Fanuc TP program (LS listing): LOWWALL.LS

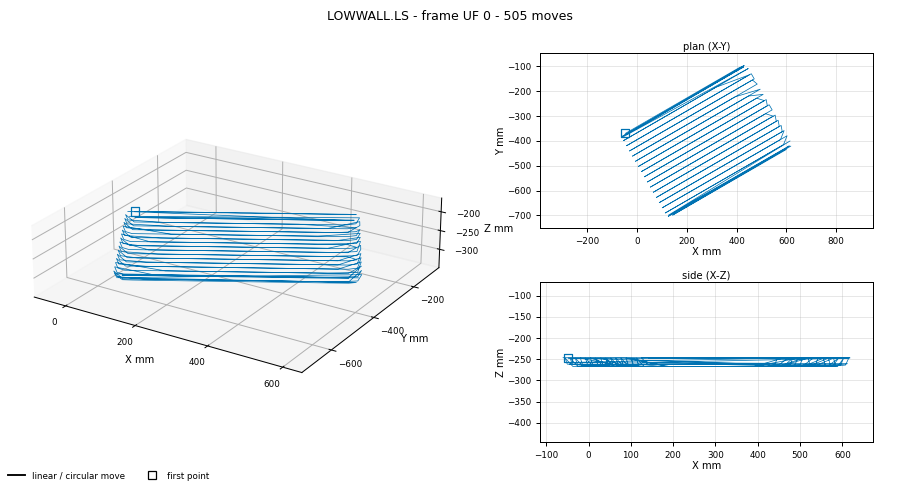
[picture p0: tool path of LOWWALL.LS in frame UF 0, 505 of 505 moves have a stored position in this frame; points joined in program order, loops and branches not executed]
/PROG  LOWWALL.LS
/ATTR
OWNER       = MNEDITOR;
COMMENT     = "";
PROG_SIZE   = 636;
CREATE      = DATE 23-01-07  TIME 11:59:14;
MODIFIED    = DATE 23-01-07  TIME 12:02:18;
FILE_NAME   = ;
VERSION     = 0;
LINE_COUNT  = 4;
MEMORY_SIZE = 992;
PROTECT     = READ_WRITE;
TCD:  STACK_SIZE	= 0,
      TASK_PRIORITY	= 50,
      TIME_SLICE	= 0,
      BUSY_LAMP_OFF	= 0,
      ABORT_REQUEST	= 0,
      PAUSE_REQUEST	= 0;
DEFAULT_GROUP	= 1,*,*,*,*;
CONTROL_CODE	= 00000000 00000000;
/MN
   1:J P[1] 100% FINE    ;
   2:L P[2] 100mm/sec CNT0    ;
   3:L P[3] 100mm/sec CNT0    ;
   4:L P[4] 100mm/sec CNT0    ;
   5:L P[5] 100mm/sec CNT0    ;
   6:L P[6] 100mm/sec CNT0    ;
   7:L P[7] 100mm/sec CNT0    ;
   8:L P[8] 100mm/sec CNT0    ;
   9:L P[9] 100mm/sec CNT0    ;
   10:L P[10] 100mm/sec CNT0    ;
   11:L P[11] 100mm/sec CNT0    ;
   12:L P[12] 100mm/sec CNT0    ;
   13:L P[13] 100mm/sec CNT0    ;
   14:L P[14] 100mm/sec CNT0    ;
   15:L P[15] 100mm/sec CNT0    ;
   16:L P[16] 100mm/sec CNT0    ;
   17:L P[17] 100mm/sec CNT0    ;
   18:L P[18] 100mm/sec CNT0    ;
   19:L P[19] 100mm/sec CNT0    ;
   20:L P[20] 100mm/sec CNT0    ;
   21:L P[21] 100mm/sec CNT0    ;
   22:L P[22] 100mm/sec CNT0    ;
   23:L P[23] 100mm/sec CNT0    ;
   24:L P[24] 100mm/sec CNT0    ;
   25:L P[25] 100mm/sec CNT0    ;
   26:L P[26] 100mm/sec CNT0    ;
   27:L P[27] 100mm/sec CNT0    ;
   28:L P[28] 100mm/sec CNT0    ;
   29:L P[29] 100mm/sec CNT0    ;
   30:L P[30] 100mm/sec CNT0    ;
   31:L P[31] 100mm/sec CNT0    ;
   32:L P[32] 100mm/sec CNT0    ;
   33:L P[33] 100mm/sec CNT0    ;
   34:L P[34] 100mm/sec CNT0    ;
   35:L P[35] 100mm/sec CNT0    ;
   36:L P[36] 100mm/sec CNT0    ;
   37:L P[37] 100mm/sec CNT0    ;
   38:L P[38] 100mm/sec CNT0    ;
   39:L P[39] 100mm/sec CNT0    ;
   40:L P[40] 100mm/sec CNT0    ;
   41:L P[41] 100mm/sec CNT0    ;
   42:L P[42] 100mm/sec CNT0    ;
   43:L P[43] 100mm/sec CNT0    ;
   44:L P[44] 100mm/sec CNT0    ;
   45:L P[45] 100mm/sec CNT0    ;
   46:L P[46] 100mm/sec CNT0    ;
   47:L P[47] 100mm/sec CNT0    ;
   48:L P[48] 100mm/sec CNT0    ;
   49:L P[49] 100mm/sec CNT0    ;
   50:L P[50] 100mm/sec CNT0    ;
   51:L P[51] 100mm/sec CNT0    ;
   52:L P[52] 100mm/sec CNT0    ;
   53:L P[53] 100mm/sec CNT0    ;
   54:L P[54] 100mm/sec CNT0    ;
   55:L P[55] 100mm/sec CNT0    ;
   56:L P[56] 100mm/sec CNT0    ;
   57:L P[57] 100mm/sec CNT0    ;
   58:L P[58] 100mm/sec CNT0    ;
   59:L P[59] 100mm/sec CNT0    ;
   60:L P[60] 100mm/sec CNT0    ;
   61:L P[61] 100mm/sec CNT0    ;
   62:L P[62] 100mm/sec CNT0    ;
   63:L P[63] 100mm/sec CNT0    ;
   64:L P[64] 100mm/sec CNT0    ;
   65:L P[65] 100mm/sec CNT0    ;
   66:L P[66] 100mm/sec CNT0    ;
   67:L P[67] 100mm/sec CNT0    ;
   68:L P[68] 100mm/sec CNT0    ;
   69:L P[69] 100mm/sec CNT0    ;
   70:L P[70] 100mm/sec CNT0    ;
   71:L P[71] 100mm/sec CNT0    ;
   72:L P[72] 100mm/sec CNT0    ;
   73:L P[73] 100mm/sec CNT0    ;
   74:L P[74] 100mm/sec CNT0    ;
   75:L P[75] 100mm/sec CNT0    ;
   76:L P[76] 100mm/sec CNT0    ;
   77:L P[77] 100mm/sec CNT0    ;
   78:L P[78] 100mm/sec CNT0    ;
   79:L P[79] 100mm/sec CNT0    ;
   80:L P[80] 100mm/sec CNT0    ;
   81:L P[81] 100mm/sec CNT0    ;
   82:L P[82] 100mm/sec CNT0    ;
   83:L P[83] 100mm/sec CNT0    ;
   84:L P[84] 100mm/sec CNT0    ;
   85:L P[85] 100mm/sec CNT0    ;
   86:L P[86] 100mm/sec CNT0    ;
   87:L P[87] 100mm/sec CNT0    ;
   88:L P[88] 100mm/sec CNT0    ;
   89:L P[89] 100mm/sec CNT0    ;
   90:L P[90] 100mm/sec CNT0    ;
   91:L P[91] 100mm/sec CNT0    ;
   92:L P[92] 100mm/sec CNT0    ;
   93:L P[93] 100mm/sec CNT0    ;
   94:L P[94] 100mm/sec CNT0    ;
   95:L P[95] 100mm/sec CNT0    ;
   96:L P[96] 100mm/sec CNT0    ;
   97:L P[97] 100mm/sec CNT0    ;
   98:L P[98] 100mm/sec CNT0    ;
   99:L P[99] 100mm/sec CNT0    ;
   100:L P[100] 100mm/sec CNT0    ;
   101:L P[101] 100mm/sec CNT0    ;
   102:L P[102] 100mm/sec CNT0    ;
   103:L P[103] 100mm/sec CNT0    ;
   104:L P[104] 100mm/sec CNT0    ;
   105:L P[105] 100mm/sec CNT0    ;
   106:L P[106] 100mm/sec CNT0    ;
   107:L P[107] 100mm/sec CNT0    ;
   108:L P[108] 100mm/sec CNT0    ;
   109:L P[109] 100mm/sec CNT0    ;
   110:L P[110] 100mm/sec CNT0    ;
   111:L P[111] 100mm/sec CNT0    ;
   112:L P[112] 100mm/sec CNT0    ;
   113:L P[113] 100mm/sec CNT0    ;
   114:L P[114] 100mm/sec CNT0    ;
   115:L P[115] 100mm/sec CNT0    ;
   116:L P[116] 100mm/sec CNT0    ;
   117:L P[117] 100mm/sec CNT0    ;
   118:L P[118] 100mm/sec CNT0    ;
   119:L P[119] 100mm/sec CNT0    ;
   120:L P[120] 100mm/sec CNT0    ;
   121:L P[121] 100mm/sec CNT0    ;
   122:L P[122] 100mm/sec CNT0    ;
   123:L P[123] 100mm/sec CNT0    ;
   124:L P[124] 100mm/sec CNT0    ;
   125:L P[125] 100mm/sec CNT0    ;
   126:L P[126] 100mm/sec CNT0    ;
   127:L P[127] 100mm/sec CNT0    ;
   128:L P[128] 100mm/sec CNT0    ;
   129:L P[129] 100mm/sec CNT0    ;
   130:L P[130] 100mm/sec CNT0    ;
   131:L P[131] 100mm/sec CNT0    ;
   132:L P[132] 100mm/sec CNT0    ;
   133:L P[133] 100mm/sec CNT0    ;
   134:L P[134] 100mm/sec CNT0    ;
   135:L P[135] 100mm/sec CNT0    ;
   136:L P[136] 100mm/sec CNT0    ;
   137:L P[137] 100mm/sec CNT0    ;
   138:L P[138] 100mm/sec CNT0    ;
   139:L P[139] 100mm/sec CNT0    ;
   140:L P[140] 100mm/sec CNT0    ;
   141:L P[141] 100mm/sec CNT0    ;
   142:L P[142] 100mm/sec CNT0    ;
   143:L P[143] 100mm/sec CNT0    ;
   144:L P[144] 100mm/sec CNT0    ;
   145:L P[145] 100mm/sec CNT0    ;
   146:L P[146] 100mm/sec CNT0    ;
   147:L P[147] 100mm/sec CNT0    ;
   148:L P[148] 100mm/sec CNT0    ;
   149:L P[149] 100mm/sec CNT0    ;
   150:L P[150] 100mm/sec CNT0    ;
   151:L P[151] 100mm/sec CNT0    ;
   152:L P[152] 100mm/sec CNT0    ;
   153:L P[153] 100mm/sec CNT0    ;
   154:L P[154] 100mm/sec CNT0    ;
   155:L P[155] 100mm/sec CNT0    ;
   156:L P[156] 100mm/sec CNT0    ;
   157:L P[157] 100mm/sec CNT0    ;
   158:L P[158] 100mm/sec CNT0    ;
   159:L P[159] 100mm/sec CNT0    ;
   160:L P[160] 100mm/sec CNT0    ;
   161:L P[161] 100mm/sec CNT0    ;
   162:L P[162] 100mm/sec CNT0    ;
   163:L P[163] 100mm/sec CNT0    ;
   164:L P[164] 100mm/sec CNT0    ;
   165:L P[165] 100mm/sec CNT0    ;
   166:L P[166] 100mm/sec CNT0    ;
   167:L P[167] 100mm/sec CNT0    ;
   168:L P[168] 100mm/sec CNT0    ;
   169:L P[169] 100mm/sec CNT0    ;
   170:L P[170] 100mm/sec CNT0    ;
   171:L P[171] 100mm/sec CNT0    ;
   172:L P[172] 100mm/sec CNT0    ;
   173:L P[173] 100mm/sec CNT0    ;
   174:L P[174] 100mm/sec CNT0    ;
   175:L P[175] 100mm/sec CNT0    ;
   176:L P[176] 100mm/sec CNT0    ;
   177:L P[177] 100mm/sec CNT0    ;
   178:L P[178] 100mm/sec CNT0    ;
   179:L P[179] 100mm/sec CNT0    ;
   180:L P[180] 100mm/sec CNT0    ;
   181:L P[181] 100mm/sec CNT0    ;
   182:L P[182] 100mm/sec CNT0    ;
   183:L P[183] 100mm/sec CNT0    ;
   184:L P[184] 100mm/sec CNT0    ;
   185:L P[185] 100mm/sec CNT0    ;
   186:L P[186] 100mm/sec CNT0    ;
   187:L P[187] 100mm/sec CNT0    ;
   188:L P[188] 100mm/sec CNT0    ;
   189:L P[189] 100mm/sec CNT0    ;
   190:L P[190] 100mm/sec CNT0    ;
   191:L P[191] 100mm/sec CNT0    ;
   192:L P[192] 100mm/sec CNT0    ;
   193:L P[193] 100mm/sec CNT0    ;
   194:L P[194] 100mm/sec CNT0    ;
   195:L P[195] 100mm/sec CNT0    ;
   196:L P[196] 100mm/sec CNT0    ;
   197:L P[197] 100mm/sec CNT0    ;
   198:L P[198] 100mm/sec CNT0    ;
   199:L P[199] 100mm/sec CNT0    ;
   200:L P[200] 100mm/sec CNT0    ;
   201:L P[201] 100mm/sec CNT0    ;
   202:L P[202] 100mm/sec CNT0    ;
   203:L P[203] 100mm/sec CNT0    ;
   204:L P[204] 100mm/sec CNT0    ;
   205:L P[205] 100mm/sec CNT0    ;
   206:L P[206] 100mm/sec CNT0    ;
   207:L P[207] 100mm/sec CNT0    ;
   208:L P[208] 100mm/sec CNT0    ;
   209:L P[209] 100mm/sec CNT0    ;
   210:L P[210] 100mm/sec CNT0    ;
   211:L P[211] 100mm/sec CNT0    ;
   212:L P[212] 100mm/sec CNT0    ;
   213:L P[213] 100mm/sec CNT0    ;
   214:L P[214] 100mm/sec CNT0    ;
   215:L P[215] 100mm/sec CNT0    ;
   216:L P[216] 100mm/sec CNT0    ;
   217:L P[217] 100mm/sec CNT0    ;
   218:L P[218] 100mm/sec CNT0    ;
   219:L P[219] 100mm/sec CNT0    ;
   220:L P[220] 100mm/sec CNT0    ;
   221:L P[221] 100mm/sec CNT0    ;
   222:L P[222] 100mm/sec CNT0    ;
   223:L P[223] 100mm/sec CNT0    ;
   224:L P[224] 100mm/sec CNT0    ;
   225:L P[225] 100mm/sec CNT0    ;
   226:L P[226] 100mm/sec CNT0    ;
   227:L P[227] 100mm/sec CNT0    ;
   228:L P[228] 100mm/sec CNT0    ;
   229:L P[229] 100mm/sec CNT0    ;
   230:L P[230] 100mm/sec CNT0    ;
   231:L P[231] 100mm/sec CNT0    ;
   232:L P[232] 100mm/sec CNT0    ;
   233:L P[233] 100mm/sec CNT0    ;
   234:L P[234] 100mm/sec CNT0    ;
   235:L P[235] 100mm/sec CNT0    ;
   236:L P[236] 100mm/sec CNT0    ;
   237:L P[237] 100mm/sec CNT0    ;
   238:L P[238] 100mm/sec CNT0    ;
   239:L P[239] 100mm/sec CNT0    ;
   240:L P[240] 100mm/sec CNT0    ;
   241:L P[241] 100mm/sec CNT0    ;
   242:L P[242] 100mm/sec CNT0    ;
   243:L P[243] 100mm/sec CNT0    ;
   244:L P[244] 100mm/sec CNT0    ;
   245:L P[245] 100mm/sec CNT0    ;
   246:L P[246] 100mm/sec CNT0    ;
   247:L P[247] 100mm/sec CNT0    ;
   248:L P[248] 100mm/sec CNT0    ;
   249:L P[249] 100mm/sec CNT0    ;
   250:L P[250] 100mm/sec CNT0    ;
   251:L P[251] 100mm/sec CNT0    ;
   252:L P[252] 100mm/sec CNT0    ;
   253:L P[253] 100mm/sec CNT0    ;
   254:L P[254] 100mm/sec CNT0    ;
   255:L P[255] 100mm/sec CNT0    ;
   256:L P[256] 100mm/sec CNT0    ;
   257:L P[257] 100mm/sec CNT0    ;
   258:L P[258] 100mm/sec CNT0    ;
   259:L P[259] 100mm/sec CNT0    ;
   260:L P[260] 100mm/sec CNT0    ;
   261:L P[261] 100mm/sec CNT0    ;
   262:L P[262] 100mm/sec CNT0    ;
   263:L P[263] 100mm/sec CNT0    ;
   264:L P[264] 100mm/sec CNT0    ;
   265:L P[265] 100mm/sec CNT0    ;
   266:L P[266] 100mm/sec CNT0    ;
   267:L P[267] 100mm/sec CNT0    ;
   268:L P[268] 100mm/sec CNT0    ;
   269:L P[269] 100mm/sec CNT0    ;
   270:L P[270] 100mm/sec CNT0    ;
   271:L P[271] 100mm/sec CNT0    ;
   272:L P[272] 100mm/sec CNT0    ;
   273:L P[273] 100mm/sec CNT0    ;
   274:L P[274] 100mm/sec CNT0    ;
   275:L P[275] 100mm/sec CNT0    ;
   276:L P[276] 100mm/sec CNT0    ;
   277:L P[277] 100mm/sec CNT0    ;
   278:L P[278] 100mm/sec CNT0    ;
   279:L P[279] 100mm/sec CNT0    ;
   280:L P[280] 100mm/sec CNT0    ;
   281:L P[281] 100mm/sec CNT0    ;
   282:L P[282] 100mm/sec CNT0    ;
   283:L P[283] 100mm/sec CNT0    ;
   284:L P[284] 100mm/sec CNT0    ;
   285:L P[285] 100mm/sec CNT0    ;
   286:L P[286] 100mm/sec CNT0    ;
   287:L P[287] 100mm/sec CNT0    ;
   288:L P[288] 100mm/sec CNT0    ;
   289:L P[289] 100mm/sec CNT0    ;
   290:L P[290] 100mm/sec CNT0    ;
   291:L P[291] 100mm/sec CNT0    ;
   292:L P[292] 100mm/sec CNT0    ;
   293:L P[293] 100mm/sec CNT0    ;
   294:L P[294] 100mm/sec CNT0    ;
   295:L P[295] 100mm/sec CNT0    ;
   296:L P[296] 100mm/sec CNT0    ;
   297:L P[297] 100mm/sec CNT0    ;
   298:L P[298] 100mm/sec CNT0    ;
   299:L P[299] 100mm/sec CNT0    ;
   300:L P[300] 100mm/sec CNT0    ;
   301:L P[301] 100mm/sec CNT0    ;
   302:L P[302] 100mm/sec CNT0    ;
   303:L P[303] 100mm/sec CNT0    ;
   304:L P[304] 100mm/sec CNT0    ;
   305:L P[305] 100mm/sec CNT0    ;
   306:L P[306] 100mm/sec CNT0    ;
   307:L P[307] 100mm/sec CNT0    ;
   308:L P[308] 100mm/sec CNT0    ;
   309:L P[309] 100mm/sec CNT0    ;
   310:L P[310] 100mm/sec CNT0    ;
   311:L P[311] 100mm/sec CNT0    ;
   312:L P[312] 100mm/sec CNT0    ;
   313:L P[313] 100mm/sec CNT0    ;
   314:L P[314] 100mm/sec CNT0    ;
   315:L P[315] 100mm/sec CNT0    ;
   316:L P[316] 100mm/sec CNT0    ;
   317:L P[317] 100mm/sec CNT0    ;
   318:L P[318] 100mm/sec CNT0    ;
   319:L P[319] 100mm/sec CNT0    ;
   320:L P[320] 100mm/sec CNT0    ;
   321:L P[321] 100mm/sec CNT0    ;
   322:L P[322] 100mm/sec CNT0    ;
   323:L P[323] 100mm/sec CNT0    ;
   324:L P[324] 100mm/sec CNT0    ;
   325:L P[325] 100mm/sec CNT0    ;
   326:L P[326] 100mm/sec CNT0    ;
   327:L P[327] 100mm/sec CNT0    ;
   328:L P[328] 100mm/sec CNT0    ;
   329:L P[329] 100mm/sec CNT0    ;
   330:L P[330] 100mm/sec CNT0    ;
   331:L P[331] 100mm/sec CNT0    ;
   332:L P[332] 100mm/sec CNT0    ;
   333:L P[333] 100mm/sec CNT0    ;
   334:L P[334] 100mm/sec CNT0    ;
   335:L P[335] 100mm/sec CNT0    ;
   336:L P[336] 100mm/sec CNT0    ;
   337:L P[337] 100mm/sec CNT0    ;
   338:L P[338] 100mm/sec CNT0    ;
   339:L P[339] 100mm/sec CNT0    ;
   340:L P[340] 100mm/sec CNT0    ;
   341:L P[341] 100mm/sec CNT0    ;
   342:L P[342] 100mm/sec CNT0    ;
   343:L P[343] 100mm/sec CNT0    ;
   344:L P[344] 100mm/sec CNT0    ;
   345:L P[345] 100mm/sec CNT0    ;
   346:L P[346] 100mm/sec CNT0    ;
   347:L P[347] 100mm/sec CNT0    ;
   348:L P[348] 100mm/sec CNT0    ;
   349:L P[349] 100mm/sec CNT0    ;
   350:L P[350] 100mm/sec CNT0    ;
   351:L P[351] 100mm/sec CNT0    ;
   352:L P[352] 100mm/sec CNT0    ;
   353:L P[353] 100mm/sec CNT0    ;
   354:L P[354] 100mm/sec CNT0    ;
   355:L P[355] 100mm/sec CNT0    ;
   356:L P[356] 100mm/sec CNT0    ;
   357:L P[357] 100mm/sec CNT0    ;
   358:L P[358] 100mm/sec CNT0    ;
   359:L P[359] 100mm/sec CNT0    ;
   360:L P[360] 100mm/sec CNT0    ;
   361:L P[361] 100mm/sec CNT0    ;
   362:L P[362] 100mm/sec CNT0    ;
   363:L P[363] 100mm/sec CNT0    ;
   364:L P[364] 100mm/sec CNT0    ;
   365:L P[365] 100mm/sec CNT0    ;
   366:L P[366] 100mm/sec CNT0    ;
   367:L P[367] 100mm/sec CNT0    ;
   368:L P[368] 100mm/sec CNT0    ;
   369:L P[369] 100mm/sec CNT0    ;
   370:L P[370] 100mm/sec CNT0    ;
   371:L P[371] 100mm/sec CNT0    ;
   372:L P[372] 100mm/sec CNT0    ;
   373:L P[373] 100mm/sec CNT0    ;
   374:L P[374] 100mm/sec CNT0    ;
   375:L P[375] 100mm/sec CNT0    ;
   376:L P[376] 100mm/sec CNT0    ;
   377:L P[377] 100mm/sec CNT0    ;
   378:L P[378] 100mm/sec CNT0    ;
   379:L P[379] 100mm/sec CNT0    ;
   380:L P[380] 100mm/sec CNT0    ;
   381:L P[381] 100mm/sec CNT0    ;
   382:L P[382] 100mm/sec CNT0    ;
   383:L P[383] 100mm/sec CNT0    ;
   384:L P[384] 100mm/sec CNT0    ;
   385:L P[385] 100mm/sec CNT0    ;
   386:L P[386] 100mm/sec CNT0    ;
   387:L P[387] 100mm/sec CNT0    ;
   388:L P[388] 100mm/sec CNT0    ;
   389:L P[389] 100mm/sec CNT0    ;
   390:L P[390] 100mm/sec CNT0    ;
   391:L P[391] 100mm/sec CNT0    ;
   392:L P[392] 100mm/sec CNT0    ;
   393:L P[393] 100mm/sec CNT0    ;
   394:L P[394] 100mm/sec CNT0    ;
   395:L P[395] 100mm/sec CNT0    ;
   396:L P[396] 100mm/sec CNT0    ;
   397:L P[397] 100mm/sec CNT0    ;
   398:L P[398] 100mm/sec CNT0    ;
   399:L P[399] 100mm/sec CNT0    ;
   400:L P[400] 100mm/sec CNT0    ;
   401:L P[401] 100mm/sec CNT0    ;
   402:L P[402] 100mm/sec CNT0    ;
   403:L P[403] 100mm/sec CNT0    ;
   404:L P[404] 100mm/sec CNT0    ;
   405:L P[405] 100mm/sec CNT0    ;
   406:L P[406] 100mm/sec CNT0    ;
   407:L P[407] 100mm/sec CNT0    ;
   408:L P[408] 100mm/sec CNT0    ;
   409:L P[409] 100mm/sec CNT0    ;
   410:L P[410] 100mm/sec CNT0    ;
   411:L P[411] 100mm/sec CNT0    ;
   412:L P[412] 100mm/sec CNT0    ;
   413:L P[413] 100mm/sec CNT0    ;
   414:L P[414] 100mm/sec CNT0    ;
   415:L P[415] 100mm/sec CNT0    ;
   416:L P[416] 100mm/sec CNT0    ;
   417:L P[417] 100mm/sec CNT0    ;
   418:L P[418] 100mm/sec CNT0    ;
   419:L P[419] 100mm/sec CNT0    ;
   420:L P[420] 100mm/sec CNT0    ;
   421:L P[421] 100mm/sec CNT0    ;
   422:L P[422] 100mm/sec CNT0    ;
   423:L P[423] 100mm/sec CNT0    ;
   424:L P[424] 100mm/sec CNT0    ;
   425:L P[425] 100mm/sec CNT0    ;
   426:L P[426] 100mm/sec CNT0    ;
   427:L P[427] 100mm/sec CNT0    ;
   428:L P[428] 100mm/sec CNT0    ;
   429:L P[429] 100mm/sec CNT0    ;
   430:L P[430] 100mm/sec CNT0    ;
   431:L P[431] 100mm/sec CNT0    ;
   432:L P[432] 100mm/sec CNT0    ;
   433:L P[433] 100mm/sec CNT0    ;
   434:L P[434] 100mm/sec CNT0    ;
   435:L P[435] 100mm/sec CNT0    ;
   436:L P[436] 100mm/sec CNT0    ;
   437:L P[437] 100mm/sec CNT0    ;
   438:L P[438] 100mm/sec CNT0    ;
   439:L P[439] 100mm/sec CNT0    ;
   440:L P[440] 100mm/sec CNT0    ;
   441:L P[441] 100mm/sec CNT0    ;
   442:L P[442] 100mm/sec CNT0    ;
   443:L P[443] 100mm/sec CNT0    ;
   444:L P[444] 100mm/sec CNT0    ;
   445:L P[445] 100mm/sec CNT0    ;
   446:L P[446] 100mm/sec CNT0    ;
   447:L P[447] 100mm/sec CNT0    ;
   448:L P[448] 100mm/sec CNT0    ;
   449:L P[449] 100mm/sec CNT0    ;
   450:L P[450] 100mm/sec CNT0    ;
   451:L P[451] 100mm/sec CNT0    ;
   452:L P[452] 100mm/sec CNT0    ;
   453:L P[453] 100mm/sec CNT0    ;
   454:L P[454] 100mm/sec CNT0    ;
   455:L P[455] 100mm/sec CNT0    ;
   456:L P[456] 100mm/sec CNT0    ;
   457:L P[457] 100mm/sec CNT0    ;
   458:L P[458] 100mm/sec CNT0    ;
   459:L P[459] 100mm/sec CNT0    ;
   460:L P[460] 100mm/sec CNT0    ;
   461:L P[461] 100mm/sec CNT0    ;
   462:L P[462] 100mm/sec CNT0    ;
   463:L P[463] 100mm/sec CNT0    ;
   464:L P[464] 100mm/sec CNT0    ;
   465:L P[465] 100mm/sec CNT0    ;
   466:L P[466] 100mm/sec CNT0    ;
   467:L P[467] 100mm/sec CNT0    ;
   468:L P[468] 100mm/sec CNT0    ;
   469:L P[469] 100mm/sec CNT0    ;
   470:L P[470] 100mm/sec CNT0    ;
   471:L P[471] 100mm/sec CNT0    ;
   472:L P[472] 100mm/sec CNT0    ;
   473:L P[473] 100mm/sec CNT0    ;
   474:L P[474] 100mm/sec CNT0    ;
   475:L P[475] 100mm/sec CNT0    ;
   476:L P[476] 100mm/sec CNT0    ;
   477:L P[477] 100mm/sec CNT0    ;
   478:L P[478] 100mm/sec CNT0    ;
   479:L P[479] 100mm/sec CNT0    ;
   480:L P[480] 100mm/sec CNT0    ;
   481:L P[481] 100mm/sec CNT0    ;
   482:L P[482] 100mm/sec CNT0    ;
   483:L P[483] 100mm/sec CNT0    ;
   484:L P[484] 100mm/sec CNT0    ;
   485:L P[485] 100mm/sec CNT0    ;
   486:L P[486] 100mm/sec CNT0    ;
   487:L P[487] 100mm/sec CNT0    ;
   488:L P[488] 100mm/sec CNT0    ;
   489:L P[489] 100mm/sec CNT0    ;
   490:L P[490] 100mm/sec CNT0    ;
   491:L P[491] 100mm/sec CNT0    ;
   492:L P[492] 100mm/sec CNT0    ;
   493:L P[493] 100mm/sec CNT0    ;
   494:L P[494] 100mm/sec CNT0    ;
   495:L P[495] 100mm/sec CNT0    ;
   496:L P[496] 100mm/sec CNT0    ;
   497:L P[497] 100mm/sec CNT0    ;
   498:L P[498] 100mm/sec CNT0    ;
   499:L P[499] 100mm/sec CNT0    ;
   500:L P[500] 100mm/sec CNT0    ;
   501:L P[501] 100mm/sec CNT0    ;
   502:L P[502] 100mm/sec CNT0    ;
   503:L P[503] 100mm/sec CNT0    ;
   504:L P[504] 100mm/sec CNT0    ;
   505:L P[505] 100mm/sec CNT0    ;
/POS
P[1]{
   GP1:
	UF : 0, UT : 6,		CONFIG : 'N U T, 0, 0, 0',
	X =  -47.550  mm,	Y =   -370.000  mm,	Z =   -247.494  mm,
	W =  90.000 deg,	P =   0.000 deg,	R =   90.000 deg
};
P[2]{
   GP1:
	UF : 0, UT : 6,		CONFIG : 'N U T, 0, 0, 0',
	X =  -26.618  mm,	Y =   -357.826  mm,	Z =   -247.507  mm,
	W =  90.000 deg,	P =   0.000 deg,	R =   90.000 deg
};
P[3]{
   GP1:
	UF : 0, UT : 6,		CONFIG : 'N U T, 0, 0, 0',
	X =  -5.744  mm,	Y =   -345.692  mm,	Z =   -247.310  mm,
	W =  90.000 deg,	P =   0.000 deg,	R =   90.000 deg
};
P[4]{
   GP1:
	UF : 0, UT : 6,		CONFIG : 'N U T, 0, 0, 0',
	X =  14.806  mm,	Y =   -333.821  mm,	Z =   -247.298  mm,
	W =  90.000 deg,	P =   0.000 deg,	R =   90.000 deg
};
P[5]{
   GP1:
	UF : 0, UT : 6,		CONFIG : 'N U T, 0, 0, 0',
	X =  35.704  mm,	Y =   -321.826  mm,	Z =   -247.469  mm,
	W =  90.000 deg,	P =   0.000 deg,	R =   90.000 deg
};
P[6]{
   GP1:
	UF : 0, UT : 6,		CONFIG : 'N U T, 0, 0, 0',
	X =  56.373  mm,	Y =   -309.892  mm,	Z =   -247.469  mm,
	W =  90.000 deg,	P =   0.000 deg,	R =   90.000 deg
};
P[7]{
   GP1:
	UF : 0, UT : 6,		CONFIG : 'N U T, 0, 0, 0',
	X =  77.152  mm,	Y =   -297.810  mm,	Z =   -247.265  mm,
	W =  90.000 deg,	P =   0.000 deg,	R =   90.000 deg
};
P[8]{
   GP1:
	UF : 0, UT : 6,		CONFIG : 'N U T, 0, 0, 0',
	X =  97.870  mm,	Y =   -285.956  mm,	Z =   -247.529  mm,
	W =  90.000 deg,	P =   0.000 deg,	R =   90.000 deg
};
P[9]{
   GP1:
	UF : 0, UT : 6,		CONFIG : 'N U T, 0, 0, 0',
	X =  118.697  mm,	Y =   -273.983  mm,	Z =   -247.655  mm,
	W =  90.000 deg,	P =   0.000 deg,	R =   90.000 deg
};
P[10]{
   GP1:
	UF : 0, UT : 6,		CONFIG : 'N U T, 0, 0, 0',
	X =  139.386  mm,	Y =   -261.886  mm,	Z =   -247.288  mm,
	W =  90.000 deg,	P =   0.000 deg,	R =   90.000 deg
};
P[11]{
   GP1:
	UF : 0, UT : 6,		CONFIG : 'N U T, 0, 0, 0',
	X =  160.242  mm,	Y =   -249.945  mm,	Z =   -247.534  mm,
	W =  90.000 deg,	P =   0.000 deg,	R =   90.000 deg
};
P[12]{
   GP1:
	UF : 0, UT : 6,		CONFIG : 'N U T, 0, 0, 0',
	X =  181.067  mm,	Y =   -237.977  mm,	Z =   -247.671  mm,
	W =  90.000 deg,	P =   0.000 deg,	R =   90.000 deg
};
P[13]{
   GP1:
	UF : 0, UT : 6,		CONFIG : 'N U T, 0, 0, 0',
	X =  202.067  mm,	Y =   -225.717  mm,	Z =   -247.343  mm,
	W =  90.000 deg,	P =   0.000 deg,	R =   90.000 deg
};
P[14]{
   GP1:
	UF : 0, UT : 6,		CONFIG : 'N U T, 0, 0, 0',
	X =  222.800  mm,	Y =   -213.811  mm,	Z =   -247.499  mm,
	W =  90.000 deg,	P =   0.000 deg,	R =   90.000 deg
};
P[15]{
   GP1:
	UF : 0, UT : 6,		CONFIG : 'N U T, 0, 0, 0',
	X =  243.481  mm,	Y =   -201.771  mm,	Z =   -247.259  mm,
	W =  90.000 deg,	P =   0.000 deg,	R =   90.000 deg
};
P[16]{
   GP1:
	UF : 0, UT : 6,		CONFIG : 'N U T, 0, 0, 0',
	X =  264.327  mm,	Y =   -189.775  mm,	Z =   -247.358  mm,
	W =  90.000 deg,	P =   0.000 deg,	R =   90.000 deg
};
P[17]{
   GP1:
	UF : 0, UT : 6,		CONFIG : 'N U T, 0, 0, 0',
	X =  284.999  mm,	Y =   -177.910  mm,	Z =   -247.531  mm,
	W =  90.000 deg,	P =   0.000 deg,	R =   90.000 deg
};
P[18]{
   GP1:
	UF : 0, UT : 6,		CONFIG : 'N U T, 0, 0, 0',
	X =  305.678  mm,	Y =   -165.935  mm,	Z =   -247.446  mm,
	W =  90.000 deg,	P =   0.000 deg,	R =   90.000 deg
};
P[19]{
   GP1:
	UF : 0, UT : 6,		CONFIG : 'N U T, 0, 0, 0',
	X =  326.574  mm,	Y =   -153.899  mm,	Z =   -247.516  mm,
	W =  90.000 deg,	P =   0.000 deg,	R =   90.000 deg
};
P[20]{
   GP1:
	UF : 0, UT : 6,		CONFIG : 'N U T, 0, 0, 0',
	X =  347.161  mm,	Y =   -142.012  mm,	Z =   -247.515  mm,
	W =  90.000 deg,	P =   0.000 deg,	R =   90.000 deg
};
P[21]{
   GP1:
	UF : 0, UT : 6,		CONFIG : 'N U T, 0, 0, 0',
	X =  368.204  mm,	Y =   -129.821  mm,	Z =   -247.414  mm,
	W =  90.000 deg,	P =   0.000 deg,	R =   90.000 deg
};
P[22]{
   GP1:
	UF : 0, UT : 6,		CONFIG : 'N U T, 0, 0, 0',
	X =  389.245  mm,	Y =   -117.683  mm,	Z =   -247.441  mm,
	W =  90.000 deg,	P =   0.000 deg,	R =   90.000 deg
};
P[23]{
   GP1:
	UF : 0, UT : 6,		CONFIG : 'N U T, 0, 0, 0',
	X =  409.743  mm,	Y =   -105.850  mm,	Z =   -247.448  mm,
	W =  90.000 deg,	P =   0.000 deg,	R =   90.000 deg
};
P[24]{
   GP1:
	UF : 0, UT : 6,		CONFIG : 'N U T, 0, 0, 0',
	X =  430.442  mm,	Y =   -96.886  mm,	Z =   -246.914  mm,
	W =  90.000 deg,	P =   0.000 deg,	R =   90.000 deg
};
P[25]{
   GP1:
	UF : 0, UT : 6,		CONFIG : 'N U T, 0, 0, 0',
	X =  -60.479  mm,	Y =   -382.088  mm,	Z =   -246.235  mm,
	W =  90.000 deg,	P =   0.000 deg,	R =   90.000 deg
};
P[26]{
   GP1:
	UF : 0, UT : 6,		CONFIG : 'N U T, 0, 0, 0',
	X =  412.489  mm,	Y =   -110.415  mm,	Z =   -261.820  mm,
	W =  90.000 deg,	P =   0.000 deg,	R =   90.000 deg
};
P[27]{
   GP1:
	UF : 0, UT : 6,		CONFIG : 'N U T, 0, 0, 0',
	X =  370.834  mm,	Y =   -134.410  mm,	Z =   -261.664  mm,
	W =  90.000 deg,	P =   0.000 deg,	R =   90.000 deg
};
P[28]{
   GP1:
	UF : 0, UT : 6,		CONFIG : 'N U T, 0, 0, 0',
	X =  350.053  mm,	Y =   -146.501  mm,	Z =   -261.826  mm,
	W =  90.000 deg,	P =   0.000 deg,	R =   90.000 deg
};
P[29]{
   GP1:
	UF : 0, UT : 6,		CONFIG : 'N U T, 0, 0, 0',
	X =  329.297  mm,	Y =   -158.443  mm,	Z =   -261.826  mm,
	W =  90.000 deg,	P =   0.000 deg,	R =   90.000 deg
};
P[30]{
   GP1:
	UF : 0, UT : 6,		CONFIG : 'N U T, 0, 0, 0',
	X =  287.613  mm,	Y =   -182.494  mm,	Z =   -261.786  mm,
	W =  90.000 deg,	P =   0.000 deg,	R =   90.000 deg
};
P[31]{
   GP1:
	UF : 0, UT : 6,		CONFIG : 'N U T, 0, 0, 0',
	X =  267.068  mm,	Y =   -194.329  mm,	Z =   -261.729  mm,
	W =  90.000 deg,	P =   0.000 deg,	R =   90.000 deg
};
P[32]{
   GP1:
	UF : 0, UT : 6,		CONFIG : 'N U T, 0, 0, 0',
	X =  246.212  mm,	Y =   -206.455  mm,	Z =   -261.878  mm,
	W =  90.000 deg,	P =   0.000 deg,	R =   90.000 deg
};
P[33]{
   GP1:
	UF : 0, UT : 6,		CONFIG : 'N U T, 0, 0, 0',
	X =  225.417  mm,	Y =   -218.435  mm,	Z =   -261.779  mm,
	W =  90.000 deg,	P =   0.000 deg,	R =   90.000 deg
};
P[34]{
   GP1:
	UF : 0, UT : 6,		CONFIG : 'N U T, 0, 0, 0',
	X =  184.036  mm,	Y =   -242.349  mm,	Z =   -261.866  mm,
	W =  90.000 deg,	P =   0.000 deg,	R =   90.000 deg
};
P[35]{
   GP1:
	UF : 0, UT : 6,		CONFIG : 'N U T, 0, 0, 0',
	X =  162.951  mm,	Y =   -254.466  mm,	Z =   -261.727  mm,
	W =  90.000 deg,	P =   0.000 deg,	R =   90.000 deg
};
P[36]{
   GP1:
	UF : 0, UT : 6,		CONFIG : 'N U T, 0, 0, 0',
	X =  142.127  mm,	Y =   -266.540  mm,	Z =   -261.832  mm,
	W =  90.000 deg,	P =   0.000 deg,	R =   90.000 deg
};
P[37]{
   GP1:
	UF : 0, UT : 6,		CONFIG : 'N U T, 0, 0, 0',
	X =  121.637  mm,	Y =   -278.384  mm,	Z =   -261.879  mm,
	W =  90.000 deg,	P =   0.000 deg,	R =   90.000 deg
};
P[38]{
   GP1:
	UF : 0, UT : 6,		CONFIG : 'N U T, 0, 0, 0',
	X =  100.557  mm,	Y =   -290.464  mm,	Z =   -261.682  mm,
	W =  90.000 deg,	P =   0.000 deg,	R =   90.000 deg
};
P[39]{
   GP1:
	UF : 0, UT : 6,		CONFIG : 'N U T, 0, 0, 0',
	X =  79.750  mm,	Y =   -302.489  mm,	Z =   -261.718  mm,
	W =  90.000 deg,	P =   0.000 deg,	R =   90.000 deg
};
P[40]{
   GP1:
	UF : 0, UT : 6,		CONFIG : 'N U T, 0, 0, 0',
	X =  59.156  mm,	Y =   -314.446  mm,	Z =   -261.818  mm,
	W =  90.000 deg,	P =   0.000 deg,	R =   90.000 deg
};
P[41]{
   GP1:
	UF : 0, UT : 6,		CONFIG : 'N U T, 0, 0, 0',
	X =  17.467  mm,	Y =   -338.426  mm,	Z =   -261.676  mm,
	W =  90.000 deg,	P =   0.000 deg,	R =   90.000 deg
};
P[42]{
   GP1:
	UF : 0, UT : 6,		CONFIG : 'N U T, 0, 0, 0',
	X =  -3.324  mm,	Y =   -350.528  mm,	Z =   -261.825  mm,
	W =  90.000 deg,	P =   0.000 deg,	R =   90.000 deg
};
P[43]{
   GP1:
	UF : 0, UT : 6,		CONFIG : 'N U T, 0, 0, 0',
	X =  -23.989  mm,	Y =   -362.468  mm,	Z =   -261.896  mm,
	W =  90.000 deg,	P =   0.000 deg,	R =   90.000 deg
};
P[44]{
   GP1:
	UF : 0, UT : 6,		CONFIG : 'N U T, 0, 0, 0',
	X =  -44.381  mm,	Y =   -374.445  mm,	Z =   -261.479  mm,
	W =  90.000 deg,	P =   0.000 deg,	R =   90.000 deg
};
P[45]{
   GP1:
	UF : 0, UT : 6,		CONFIG : 'N U T, 0, 0, 0',
	X =  38.415  mm,	Y =   -326.502  mm,	Z =   -262.006  mm,
	W =  90.000 deg,	P =   0.000 deg,	R =   90.000 deg
};
P[46]{
   GP1:
	UF : 0, UT : 6,		CONFIG : 'N U T, 0, 0, 0',
	X =  204.449  mm,	Y =   -230.596  mm,	Z =   -261.901  mm,
	W =  90.000 deg,	P =   0.000 deg,	R =   90.000 deg
};
P[47]{
   GP1:
	UF : 0, UT : 6,		CONFIG : 'N U T, 0, 0, 0',
	X =  308.404  mm,	Y =   -170.556  mm,	Z =   -261.891  mm,
	W =  90.000 deg,	P =   0.000 deg,	R =   90.000 deg
};
P[48]{
   GP1:
	UF : 0, UT : 6,		CONFIG : 'N U T, 0, 0, 0',
	X =  391.691  mm,	Y =   -122.489  mm,	Z =   -261.923  mm,
	W =  90.000 deg,	P =   0.000 deg,	R =   90.000 deg
};
P[49]{
   GP1:
	UF : 0, UT : 6,		CONFIG : 'N U T, 0, 0, 0',
	X =  428.244  mm,	Y =   -102.644  mm,	Z =   -260.471  mm,
	W =  90.000 deg,	P =   0.000 deg,	R =   90.000 deg
};
P[50]{
   GP1:
	UF : 0, UT : 6,		CONFIG : 'N U T, 0, 0, 0',
	X =  -55.260  mm,	Y =   -383.192  mm,	Z =   -257.735  mm,
	W =  90.000 deg,	P =   0.000 deg,	R =   90.000 deg
};
P[51]{
   GP1:
	UF : 0, UT : 6,		CONFIG : 'N U T, 0, 0, 0',
	X =  446.546  mm,	Y =   -108.963  mm,	Z =   -247.498  mm,
	W =  90.000 deg,	P =   0.000 deg,	R =   90.000 deg
};
P[52]{
   GP1:
	UF : 0, UT : 6,		CONFIG : 'N U T, 0, 0, 0',
	X =  439.168  mm,	Y =   -113.350  mm,	Z =   -263.581  mm,
	W =  90.000 deg,	P =   0.000 deg,	R =   90.000 deg
};
P[53]{
   GP1:
	UF : 0, UT : 6,		CONFIG : 'N U T, 0, 0, 0',
	X =  420.370  mm,	Y =   -124.132  mm,	Z =   -267.000  mm,
	W =  90.000 deg,	P =   0.000 deg,	R =   90.000 deg
};
P[54]{
   GP1:
	UF : 0, UT : 6,		CONFIG : 'N U T, 0, 0, 0',
	X =  399.764  mm,	Y =   -136.182  mm,	Z =   -267.000  mm,
	W =  90.000 deg,	P =   0.000 deg,	R =   90.000 deg
};
P[55]{
   GP1:
	UF : 0, UT : 6,		CONFIG : 'N U T, 0, 0, 0',
	X =  378.865  mm,	Y =   -148.307  mm,	Z =   -267.000  mm,
	W =  90.000 deg,	P =   0.000 deg,	R =   90.000 deg
};
P[56]{
   GP1:
	UF : 0, UT : 6,		CONFIG : 'N U T, 0, 0, 0',
	X =  358.130  mm,	Y =   -160.268  mm,	Z =   -267.000  mm,
	W =  90.000 deg,	P =   0.000 deg,	R =   90.000 deg
};
P[57]{
   GP1:
	UF : 0, UT : 6,		CONFIG : 'N U T, 0, 0, 0',
	X =  337.379  mm,	Y =   -172.204  mm,	Z =   -267.000  mm,
	W =  90.000 deg,	P =   0.000 deg,	R =   90.000 deg
};
P[58]{
   GP1:
	UF : 0, UT : 6,		CONFIG : 'N U T, 0, 0, 0',
	X =  295.656  mm,	Y =   -196.318  mm,	Z =   -267.000  mm,
	W =  90.000 deg,	P =   0.000 deg,	R =   90.000 deg
};
P[59]{
   GP1:
	UF : 0, UT : 6,		CONFIG : 'N U T, 0, 0, 0',
	X =  254.258  mm,	Y =   -220.242  mm,	Z =   -267.000  mm,
	W =  90.000 deg,	P =   0.000 deg,	R =   90.000 deg
};
P[60]{
   GP1:
	UF : 0, UT : 6,		CONFIG : 'N U T, 0, 0, 0',
	X =  233.188  mm,	Y =   -232.339  mm,	Z =   -267.000  mm,
	W =  90.000 deg,	P =   0.000 deg,	R =   90.000 deg
};
P[61]{
   GP1:
	UF : 0, UT : 6,		CONFIG : 'N U T, 0, 0, 0',
	X =  212.591  mm,	Y =   -244.258  mm,	Z =   -267.000  mm,
	W =  90.000 deg,	P =   0.000 deg,	R =   90.000 deg
};
P[62]{
   GP1:
	UF : 0, UT : 6,		CONFIG : 'N U T, 0, 0, 0',
	X =  191.779  mm,	Y =   -256.362  mm,	Z =   -267.000  mm,
	W =  90.000 deg,	P =   0.000 deg,	R =   90.000 deg
};
P[63]{
   GP1:
	UF : 0, UT : 6,		CONFIG : 'N U T, 0, 0, 0',
	X =  150.236  mm,	Y =   -280.241  mm,	Z =   -267.000  mm,
	W =  90.000 deg,	P =   0.000 deg,	R =   90.000 deg
};
P[64]{
   GP1:
	UF : 0, UT : 6,		CONFIG : 'N U T, 0, 0, 0',
	X =  129.497  mm,	Y =   -292.201  mm,	Z =   -267.000  mm,
	W =  90.000 deg,	P =   0.000 deg,	R =   90.000 deg
};
P[65]{
   GP1:
	UF : 0, UT : 6,		CONFIG : 'N U T, 0, 0, 0',
	X =  108.608  mm,	Y =   -304.247  mm,	Z =   -267.000  mm,
	W =  90.000 deg,	P =   0.000 deg,	R =   90.000 deg
};
P[66]{
   GP1:
	UF : 0, UT : 6,		CONFIG : 'N U T, 0, 0, 0',
	X =  87.672  mm,	Y =   -316.136  mm,	Z =   -267.000  mm,
	W =  90.000 deg,	P =   0.000 deg,	R =   90.000 deg
};
P[67]{
   GP1:
	UF : 0, UT : 6,		CONFIG : 'N U T, 0, 0, 0',
	X =  46.208  mm,	Y =   -340.367  mm,	Z =   -267.000  mm,
	W =  90.000 deg,	P =   0.000 deg,	R =   90.000 deg
};
P[68]{
   GP1:
	UF : 0, UT : 6,		CONFIG : 'N U T, 0, 0, 0',
	X =  4.872  mm,	Y =   -364.275  mm,	Z =   -267.000  mm,
	W =  90.000 deg,	P =   0.000 deg,	R =   90.000 deg
};
P[69]{
   GP1:
	UF : 0, UT : 6,		CONFIG : 'N U T, 0, 0, 0',
	X =  -16.012  mm,	Y =   -376.260  mm,	Z =   -267.000  mm,
	W =  90.000 deg,	P =   0.000 deg,	R =   90.000 deg
};
P[70]{
   GP1:
	UF : 0, UT : 6,		CONFIG : 'N U T, 0, 0, 0',
	X =  -37.068  mm,	Y =   -388.355  mm,	Z =   -266.951  mm,
	W =  90.000 deg,	P =   0.000 deg,	R =   90.000 deg
};
P[71]{
   GP1:
	UF : 0, UT : 6,		CONFIG : 'N U T, 0, 0, 0',
	X =  -55.221  mm,	Y =   -398.977  mm,	Z =   -247.406  mm,
	W =  90.000 deg,	P =   0.000 deg,	R =   90.000 deg
};
P[72]{
   GP1:
	UF : 0, UT : 6,		CONFIG : 'N U T, 0, 0, 0',
	X =  -50.332  mm,	Y =   -396.514  mm,	Z =   -261.436  mm,
	W =  90.000 deg,	P =   0.000 deg,	R =   90.000 deg
};
P[73]{
   GP1:
	UF : 0, UT : 6,		CONFIG : 'N U T, 0, 0, 0',
	X =  25.566  mm,	Y =   -352.401  mm,	Z =   -267.000  mm,
	W =  90.000 deg,	P =   0.000 deg,	R =   90.000 deg
};
P[74]{
   GP1:
	UF : 0, UT : 6,		CONFIG : 'N U T, 0, 0, 0',
	X =  67.197  mm,	Y =   -328.433  mm,	Z =   -267.000  mm,
	W =  90.000 deg,	P =   0.000 deg,	R =   90.000 deg
};
P[75]{
   GP1:
	UF : 0, UT : 6,		CONFIG : 'N U T, 0, 0, 0',
	X =  170.941  mm,	Y =   -268.423  mm,	Z =   -267.000  mm,
	W =  90.000 deg,	P =   0.000 deg,	R =   90.000 deg
};
P[76]{
   GP1:
	UF : 0, UT : 6,		CONFIG : 'N U T, 0, 0, 0',
	X =  274.930  mm,	Y =   -208.442  mm,	Z =   -267.000  mm,
	W =  90.000 deg,	P =   0.000 deg,	R =   90.000 deg
};
P[77]{
   GP1:
	UF : 0, UT : 6,		CONFIG : 'N U T, 0, 0, 0',
	X =  316.669  mm,	Y =   -184.325  mm,	Z =   -267.000  mm,
	W =  90.000 deg,	P =   0.000 deg,	R =   90.000 deg
};
P[78]{
   GP1:
	UF : 0, UT : 6,		CONFIG : 'N U T, 0, 0, 0',
	X =  451.381  mm,	Y =   -134.062  mm,	Z =   -263.711  mm,
	W =  90.000 deg,	P =   0.000 deg,	R =   90.000 deg
};
P[79]{
   GP1:
	UF : 0, UT : 6,		CONFIG : 'N U T, 0, 0, 0',
	X =  432.359  mm,	Y =   -144.999  mm,	Z =   -267.000  mm,
	W =  90.000 deg,	P =   0.000 deg,	R =   90.000 deg
};
P[80]{
   GP1:
	UF : 0, UT : 6,		CONFIG : 'N U T, 0, 0, 0',
	X =  411.585  mm,	Y =   -157.094  mm,	Z =   -267.000  mm,
	W =  90.000 deg,	P =   0.000 deg,	R =   90.000 deg
};
P[81]{
   GP1:
	UF : 0, UT : 6,		CONFIG : 'N U T, 0, 0, 0',
	X =  349.418  mm,	Y =   -192.998  mm,	Z =   -267.000  mm,
	W =  90.000 deg,	P =   0.000 deg,	R =   90.000 deg
};
P[82]{
   GP1:
	UF : 0, UT : 6,		CONFIG : 'N U T, 0, 0, 0',
	X =  328.317  mm,	Y =   -204.987  mm,	Z =   -267.000  mm,
	W =  90.000 deg,	P =   0.000 deg,	R =   90.000 deg
};
P[83]{
   GP1:
	UF : 0, UT : 6,		CONFIG : 'N U T, 0, 0, 0',
	X =  307.881  mm,	Y =   -217.039  mm,	Z =   -267.000  mm,
	W =  90.000 deg,	P =   0.000 deg,	R =   90.000 deg
};
P[84]{
   GP1:
	UF : 0, UT : 6,		CONFIG : 'N U T, 0, 0, 0',
	X =  183.024  mm,	Y =   -288.927  mm,	Z =   -267.000  mm,
	W =  90.000 deg,	P =   0.000 deg,	R =   90.000 deg
};
P[85]{
   GP1:
	UF : 0, UT : 6,		CONFIG : 'N U T, 0, 0, 0',
	X =  162.128  mm,	Y =   -301.040  mm,	Z =   -267.000  mm,
	W =  90.000 deg,	P =   0.000 deg,	R =   90.000 deg
};
P[86]{
   GP1:
	UF : 0, UT : 6,		CONFIG : 'N U T, 0, 0, 0',
	X =  99.786  mm,	Y =   -336.939  mm,	Z =   -267.000  mm,
	W =  90.000 deg,	P =   0.000 deg,	R =   90.000 deg
};
P[87]{
   GP1:
	UF : 0, UT : 6,		CONFIG : 'N U T, 0, 0, 0',
	X =  37.572  mm,	Y =   -373.058  mm,	Z =   -267.000  mm,
	W =  90.000 deg,	P =   0.000 deg,	R =   90.000 deg
};
P[88]{
   GP1:
	UF : 0, UT : 6,		CONFIG : 'N U T, 0, 0, 0',
	X =  16.721  mm,	Y =   -384.953  mm,	Z =   -267.000  mm,
	W =  90.000 deg,	P =   0.000 deg,	R =   90.000 deg
};
P[89]{
   GP1:
	UF : 0, UT : 6,		CONFIG : 'N U T, 0, 0, 0',
	X =  -4.151  mm,	Y =   -397.089  mm,	Z =   -267.000  mm,
	W =  90.000 deg,	P =   0.000 deg,	R =   90.000 deg
};
P[90]{
   GP1:
	UF : 0, UT : 6,		CONFIG : 'N U T, 0, 0, 0',
	X =  -24.791  mm,	Y =   -409.044  mm,	Z =   -267.000  mm,
	W =  90.000 deg,	P =   0.000 deg,	R =   90.000 deg
};
P[91]{
   GP1:
	UF : 0, UT : 6,		CONFIG : 'N U T, 0, 0, 0',
	X =  -43.351  mm,	Y =   -419.573  mm,	Z =   -247.586  mm,
	W =  90.000 deg,	P =   0.000 deg,	R =   90.000 deg
};
P[92]{
   GP1:
	UF : 0, UT : 6,		CONFIG : 'N U T, 0, 0, 0',
	X =  -38.522  mm,	Y =   -417.253  mm,	Z =   -261.946  mm,
	W =  90.000 deg,	P =   0.000 deg,	R =   90.000 deg
};
P[93]{
   GP1:
	UF : 0, UT : 6,		CONFIG : 'N U T, 0, 0, 0',
	X =  58.534  mm,	Y =   -361.056  mm,	Z =   -267.000  mm,
	W =  90.000 deg,	P =   0.000 deg,	R =   90.000 deg
};
P[94]{
   GP1:
	UF : 0, UT : 6,		CONFIG : 'N U T, 0, 0, 0',
	X =  79.100  mm,	Y =   -349.269  mm,	Z =   -267.000  mm,
	W =  90.000 deg,	P =   0.000 deg,	R =   90.000 deg
};
P[95]{
   GP1:
	UF : 0, UT : 6,		CONFIG : 'N U T, 0, 0, 0',
	X =  120.716  mm,	Y =   -325.116  mm,	Z =   -267.000  mm,
	W =  90.000 deg,	P =   0.000 deg,	R =   90.000 deg
};
P[96]{
   GP1:
	UF : 0, UT : 6,		CONFIG : 'N U T, 0, 0, 0',
	X =  141.397  mm,	Y =   -313.254  mm,	Z =   -267.000  mm,
	W =  90.000 deg,	P =   0.000 deg,	R =   90.000 deg
};
P[97]{
   GP1:
	UF : 0, UT : 6,		CONFIG : 'N U T, 0, 0, 0',
	X =  203.954  mm,	Y =   -277.374  mm,	Z =   -267.000  mm,
	W =  90.000 deg,	P =   0.000 deg,	R =   90.000 deg
};
P[98]{
   GP1:
	UF : 0, UT : 6,		CONFIG : 'N U T, 0, 0, 0',
	X =  224.509  mm,	Y =   -265.184  mm,	Z =   -267.000  mm,
	W =  90.000 deg,	P =   0.000 deg,	R =   90.000 deg
};
P[99]{
   GP1:
	UF : 0, UT : 6,		CONFIG : 'N U T, 0, 0, 0',
	X =  245.643  mm,	Y =   -253.141  mm,	Z =   -267.000  mm,
	W =  90.000 deg,	P =   0.000 deg,	R =   90.000 deg
};
P[100]{
   GP1:
	UF : 0, UT : 6,		CONFIG : 'N U T, 0, 0, 0',
	X =  266.269  mm,	Y =   -241.146  mm,	Z =   -267.000  mm,
	W =  90.000 deg,	P =   0.000 deg,	R =   90.000 deg
};
P[101]{
   GP1:
	UF : 0, UT : 6,		CONFIG : 'N U T, 0, 0, 0',
	X =  286.852  mm,	Y =   -229.271  mm,	Z =   -267.000  mm,
	W =  90.000 deg,	P =   0.000 deg,	R =   90.000 deg
};
P[102]{
   GP1:
	UF : 0, UT : 6,		CONFIG : 'N U T, 0, 0, 0',
	X =  370.087  mm,	Y =   -181.139  mm,	Z =   -267.000  mm,
	W =  90.000 deg,	P =   0.000 deg,	R =   90.000 deg
};
P[103]{
   GP1:
	UF : 0, UT : 6,		CONFIG : 'N U T, 0, 0, 0',
	X =  390.770  mm,	Y =   -169.245  mm,	Z =   -267.000  mm,
	W =  90.000 deg,	P =   0.000 deg,	R =   90.000 deg
};
P[104]{
   GP1:
	UF : 0, UT : 6,		CONFIG : 'N U T, 0, 0, 0',
	X =  458.817  mm,	Y =   -129.922  mm,	Z =   -247.329  mm,
	W =  90.000 deg,	P =   0.000 deg,	R =   90.000 deg
};
P[105]{
   GP1:
	UF : 0, UT : 6,		CONFIG : 'N U T, 0, 0, 0',
	X =  470.747  mm,	Y =   -150.689  mm,	Z =   -247.477  mm,
	W =  90.000 deg,	P =   0.000 deg,	R =   90.000 deg
};
P[106]{
   GP1:
	UF : 0, UT : 6,		CONFIG : 'N U T, 0, 0, 0',
	X =  444.533  mm,	Y =   -165.763  mm,	Z =   -267.000  mm,
	W =  90.000 deg,	P =   0.000 deg,	R =   90.000 deg
};
P[107]{
   GP1:
	UF : 0, UT : 6,		CONFIG : 'N U T, 0, 0, 0',
	X =  402.701  mm,	Y =   -189.872  mm,	Z =   -267.000  mm,
	W =  90.000 deg,	P =   0.000 deg,	R =   90.000 deg
};
P[108]{
   GP1:
	UF : 0, UT : 6,		CONFIG : 'N U T, 0, 0, 0',
	X =  381.964  mm,	Y =   -201.832  mm,	Z =   -267.000  mm,
	W =  90.000 deg,	P =   0.000 deg,	R =   90.000 deg
};
P[109]{
   GP1:
	UF : 0, UT : 6,		CONFIG : 'N U T, 0, 0, 0',
	X =  361.394  mm,	Y =   -213.854  mm,	Z =   -267.000  mm,
	W =  90.000 deg,	P =   0.000 deg,	R =   90.000 deg
};
P[110]{
   GP1:
	UF : 0, UT : 6,		CONFIG : 'N U T, 0, 0, 0',
	X =  340.522  mm,	Y =   -225.902  mm,	Z =   -267.000  mm,
	W =  90.000 deg,	P =   0.000 deg,	R =   90.000 deg
};
P[111]{
   GP1:
	UF : 0, UT : 6,		CONFIG : 'N U T, 0, 0, 0',
	X =  319.713  mm,	Y =   -237.916  mm,	Z =   -267.000  mm,
	W =  90.000 deg,	P =   0.000 deg,	R =   90.000 deg
};
P[112]{
   GP1:
	UF : 0, UT : 6,		CONFIG : 'N U T, 0, 0, 0',
	X =  195.126  mm,	Y =   -309.790  mm,	Z =   -267.000  mm,
	W =  90.000 deg,	P =   0.000 deg,	R =   90.000 deg
};
P[113]{
   GP1:
	UF : 0, UT : 6,		CONFIG : 'N U T, 0, 0, 0',
	X =  174.289  mm,	Y =   -321.730  mm,	Z =   -267.000  mm,
	W =  90.000 deg,	P =   0.000 deg,	R =   90.000 deg
};
P[114]{
   GP1:
	UF : 0, UT : 6,		CONFIG : 'N U T, 0, 0, 0',
	X =  132.477  mm,	Y =   -345.799  mm,	Z =   -267.000  mm,
	W =  90.000 deg,	P =   0.000 deg,	R =   90.000 deg
};
P[115]{
   GP1:
	UF : 0, UT : 6,		CONFIG : 'N U T, 0, 0, 0',
	X =  111.896  mm,	Y =   -357.839  mm,	Z =   -267.000  mm,
	W =  90.000 deg,	P =   0.000 deg,	R =   90.000 deg
};
P[116]{
   GP1:
	UF : 0, UT : 6,		CONFIG : 'N U T, 0, 0, 0',
	X =  70.293  mm,	Y =   -381.797  mm,	Z =   -267.000  mm,
	W =  90.000 deg,	P =   0.000 deg,	R =   90.000 deg
};
P[117]{
   GP1:
	UF : 0, UT : 6,		CONFIG : 'N U T, 0, 0, 0',
	X =  7.939  mm,	Y =   -417.904  mm,	Z =   -267.000  mm,
	W =  90.000 deg,	P =   0.000 deg,	R =   90.000 deg
};
P[118]{
   GP1:
	UF : 0, UT : 6,		CONFIG : 'N U T, 0, 0, 0',
	X =  -12.787  mm,	Y =   -429.740  mm,	Z =   -267.000  mm,
	W =  90.000 deg,	P =   0.000 deg,	R =   90.000 deg
};
P[119]{
   GP1:
	UF : 0, UT : 6,		CONFIG : 'N U T, 0, 0, 0',
	X =  -31.205  mm,	Y =   -440.645  mm,	Z =   -247.535  mm,
	W =  90.000 deg,	P =   0.000 deg,	R =   90.000 deg
};
P[120]{
   GP1:
	UF : 0, UT : 6,		CONFIG : 'N U T, 0, 0, 0',
	X =  -26.628  mm,	Y =   -437.928  mm,	Z =   -261.889  mm,
	W =  90.000 deg,	P =   0.000 deg,	R =   90.000 deg
};
P[121]{
   GP1:
	UF : 0, UT : 6,		CONFIG : 'N U T, 0, 0, 0',
	X =  28.646  mm,	Y =   -406.067  mm,	Z =   -267.000  mm,
	W =  90.000 deg,	P =   0.000 deg,	R =   90.000 deg
};
P[122]{
   GP1:
	UF : 0, UT : 6,		CONFIG : 'N U T, 0, 0, 0',
	X =  49.813  mm,	Y =   -394.102  mm,	Z =   -267.000  mm,
	W =  90.000 deg,	P =   0.000 deg,	R =   90.000 deg
};
P[123]{
   GP1:
	UF : 0, UT : 6,		CONFIG : 'N U T, 0, 0, 0',
	X =  91.185  mm,	Y =   -369.881  mm,	Z =   -267.000  mm,
	W =  90.000 deg,	P =   0.000 deg,	R =   90.000 deg
};
P[124]{
   GP1:
	UF : 0, UT : 6,		CONFIG : 'N U T, 0, 0, 0',
	X =  153.456  mm,	Y =   -334.006  mm,	Z =   -267.000  mm,
	W =  90.000 deg,	P =   0.000 deg,	R =   90.000 deg
};
P[125]{
   GP1:
	UF : 0, UT : 6,		CONFIG : 'N U T, 0, 0, 0',
	X =  215.988  mm,	Y =   -297.950  mm,	Z =   -267.000  mm,
	W =  90.000 deg,	P =   0.000 deg,	R =   90.000 deg
};
P[126]{
   GP1:
	UF : 0, UT : 6,		CONFIG : 'N U T, 0, 0, 0',
	X =  236.863  mm,	Y =   -285.802  mm,	Z =   -267.000  mm,
	W =  90.000 deg,	P =   0.000 deg,	R =   90.000 deg
};
P[127]{
   GP1:
	UF : 0, UT : 6,		CONFIG : 'N U T, 0, 0, 0',
	X =  257.744  mm,	Y =   -273.961  mm,	Z =   -267.000  mm,
	W =  90.000 deg,	P =   0.000 deg,	R =   90.000 deg
};
P[128]{
   GP1:
	UF : 0, UT : 6,		CONFIG : 'N U T, 0, 0, 0',
	X =  278.154  mm,	Y =   -261.962  mm,	Z =   -267.000  mm,
	W =  90.000 deg,	P =   0.000 deg,	R =   90.000 deg
};
P[129]{
   GP1:
	UF : 0, UT : 6,		CONFIG : 'N U T, 0, 0, 0',
	X =  299.027  mm,	Y =   -249.939  mm,	Z =   -267.000  mm,
	W =  90.000 deg,	P =   0.000 deg,	R =   90.000 deg
};
P[130]{
   GP1:
	UF : 0, UT : 6,		CONFIG : 'N U T, 0, 0, 0',
	X =  423.689  mm,	Y =   -178.055  mm,	Z =   -267.000  mm,
	W =  90.000 deg,	P =   0.000 deg,	R =   90.000 deg
};
P[131]{
   GP1:
	UF : 0, UT : 6,		CONFIG : 'N U T, 0, 0, 0',
	X =  463.463  mm,	Y =   -155.052  mm,	Z =   -263.814  mm,
	W =  90.000 deg,	P =   0.000 deg,	R =   90.000 deg
};
P[132]{
   GP1:
	UF : 0, UT : 6,		CONFIG : 'N U T, 0, 0, 0',
	X =  482.747  mm,	Y =   -171.485  mm,	Z =   -247.497  mm,
	W =  90.000 deg,	P =   0.000 deg,	R =   90.000 deg
};
P[133]{
   GP1:
	UF : 0, UT : 6,		CONFIG : 'N U T, 0, 0, 0',
	X =  475.285  mm,	Y =   -175.809  mm,	Z =   -263.860  mm,
	W =  90.000 deg,	P =   0.000 deg,	R =   90.000 deg
};
P[134]{
   GP1:
	UF : 0, UT : 6,		CONFIG : 'N U T, 0, 0, 0',
	X =  456.233  mm,	Y =   -186.509  mm,	Z =   -267.000  mm,
	W =  90.000 deg,	P =   0.000 deg,	R =   90.000 deg
};
P[135]{
   GP1:
	UF : 0, UT : 6,		CONFIG : 'N U T, 0, 0, 0',
	X =  435.634  mm,	Y =   -198.578  mm,	Z =   -267.000  mm,
	W =  90.000 deg,	P =   0.000 deg,	R =   90.000 deg
};
P[136]{
   GP1:
	UF : 0, UT : 6,		CONFIG : 'N U T, 0, 0, 0',
	X =  414.827  mm,	Y =   -210.721  mm,	Z =   -267.000  mm,
	W =  90.000 deg,	P =   0.000 deg,	R =   90.000 deg
};
P[137]{
   GP1:
	UF : 0, UT : 6,		CONFIG : 'N U T, 0, 0, 0',
	X =  373.256  mm,	Y =   -234.506  mm,	Z =   -267.000  mm,
	W =  90.000 deg,	P =   0.000 deg,	R =   90.000 deg
};
P[138]{
   GP1:
	UF : 0, UT : 6,		CONFIG : 'N U T, 0, 0, 0',
	X =  352.463  mm,	Y =   -246.699  mm,	Z =   -267.000  mm,
	W =  90.000 deg,	P =   0.000 deg,	R =   90.000 deg
};
P[139]{
   GP1:
	UF : 0, UT : 6,		CONFIG : 'N U T, 0, 0, 0',
	X =  311.047  mm,	Y =   -270.622  mm,	Z =   -267.000  mm,
	W =  90.000 deg,	P =   0.000 deg,	R =   90.000 deg
};
P[140]{
   GP1:
	UF : 0, UT : 6,		CONFIG : 'N U T, 0, 0, 0',
	X =  289.985  mm,	Y =   -282.694  mm,	Z =   -267.000  mm,
	W =  90.000 deg,	P =   0.000 deg,	R =   90.000 deg
};
P[141]{
   GP1:
	UF : 0, UT : 6,		CONFIG : 'N U T, 0, 0, 0',
	X =  248.426  mm,	Y =   -306.749  mm,	Z =   -267.000  mm,
	W =  90.000 deg,	P =   0.000 deg,	R =   90.000 deg
};
P[142]{
   GP1:
	UF : 0, UT : 6,		CONFIG : 'N U T, 0, 0, 0',
	X =  227.947  mm,	Y =   -318.512  mm,	Z =   -267.000  mm,
	W =  90.000 deg,	P =   0.000 deg,	R =   90.000 deg
};
P[143]{
   GP1:
	UF : 0, UT : 6,		CONFIG : 'N U T, 0, 0, 0',
	X =  186.069  mm,	Y =   -342.692  mm,	Z =   -267.000  mm,
	W =  90.000 deg,	P =   0.000 deg,	R =   90.000 deg
};
P[144]{
   GP1:
	UF : 0, UT : 6,		CONFIG : 'N U T, 0, 0, 0',
	X =  165.362  mm,	Y =   -354.747  mm,	Z =   -267.000  mm,
	W =  90.000 deg,	P =   0.000 deg,	R =   90.000 deg
};
P[145]{
   GP1:
	UF : 0, UT : 6,		CONFIG : 'N U T, 0, 0, 0',
	X =  144.582  mm,	Y =   -366.659  mm,	Z =   -267.000  mm,
	W =  90.000 deg,	P =   0.000 deg,	R =   90.000 deg
};
P[146]{
   GP1:
	UF : 0, UT : 6,		CONFIG : 'N U T, 0, 0, 0',
	X =  123.865  mm,	Y =   -378.675  mm,	Z =   -267.000  mm,
	W =  90.000 deg,	P =   0.000 deg,	R =   90.000 deg
};
P[147]{
   GP1:
	UF : 0, UT : 6,		CONFIG : 'N U T, 0, 0, 0',
	X =  103.206  mm,	Y =   -390.534  mm,	Z =   -267.000  mm,
	W =  90.000 deg,	P =   0.000 deg,	R =   90.000 deg
};
P[148]{
   GP1:
	UF : 0, UT : 6,		CONFIG : 'N U T, 0, 0, 0',
	X =  61.476  mm,	Y =   -414.721  mm,	Z =   -267.000  mm,
	W =  90.000 deg,	P =   0.000 deg,	R =   90.000 deg
};
P[149]{
   GP1:
	UF : 0, UT : 6,		CONFIG : 'N U T, 0, 0, 0',
	X =  40.701  mm,	Y =   -426.420  mm,	Z =   -267.000  mm,
	W =  90.000 deg,	P =   0.000 deg,	R =   90.000 deg
};
P[150]{
   GP1:
	UF : 0, UT : 6,		CONFIG : 'N U T, 0, 0, 0',
	X =  19.908  mm,	Y =   -438.743  mm,	Z =   -267.000  mm,
	W =  90.000 deg,	P =   0.000 deg,	R =   90.000 deg
};
P[151]{
   GP1:
	UF : 0, UT : 6,		CONFIG : 'N U T, 0, 0, 0',
	X =  -0.866  mm,	Y =   -450.609  mm,	Z =   -267.000  mm,
	W =  90.000 deg,	P =   0.000 deg,	R =   90.000 deg
};
P[152]{
   GP1:
	UF : 0, UT : 6,		CONFIG : 'N U T, 0, 0, 0',
	X =  -14.744  mm,	Y =   -458.593  mm,	Z =   -261.769  mm,
	W =  90.000 deg,	P =   0.000 deg,	R =   90.000 deg
};
P[153]{
   GP1:
	UF : 0, UT : 6,		CONFIG : 'N U T, 0, 0, 0',
	X =  -19.252  mm,	Y =   -461.476  mm,	Z =   -247.354  mm,
	W =  90.000 deg,	P =   0.000 deg,	R =   90.000 deg
};
P[154]{
   GP1:
	UF : 0, UT : 6,		CONFIG : 'N U T, 0, 0, 0',
	X =  82.632  mm,	Y =   -402.728  mm,	Z =   -267.000  mm,
	W =  90.000 deg,	P =   0.000 deg,	R =   90.000 deg
};
P[155]{
   GP1:
	UF : 0, UT : 6,		CONFIG : 'N U T, 0, 0, 0',
	X =  207.189  mm,	Y =   -330.649  mm,	Z =   -267.000  mm,
	W =  90.000 deg,	P =   0.000 deg,	R =   90.000 deg
};
P[156]{
   GP1:
	UF : 0, UT : 6,		CONFIG : 'N U T, 0, 0, 0',
	X =  269.546  mm,	Y =   -294.778  mm,	Z =   -267.000  mm,
	W =  90.000 deg,	P =   0.000 deg,	R =   90.000 deg
};
P[157]{
   GP1:
	UF : 0, UT : 6,		CONFIG : 'N U T, 0, 0, 0',
	X =  332.038  mm,	Y =   -258.753  mm,	Z =   -267.000  mm,
	W =  90.000 deg,	P =   0.000 deg,	R =   90.000 deg
};
P[158]{
   GP1:
	UF : 0, UT : 6,		CONFIG : 'N U T, 0, 0, 0',
	X =  394.050  mm,	Y =   -222.762  mm,	Z =   -267.000  mm,
	W =  90.000 deg,	P =   0.000 deg,	R =   90.000 deg
};
P[159]{
   GP1:
	UF : 0, UT : 6,		CONFIG : 'N U T, 0, 0, 0',
	X =  494.735  mm,	Y =   -192.184  mm,	Z =   -247.407  mm,
	W =  90.000 deg,	P =   0.000 deg,	R =   90.000 deg
};
P[160]{
   GP1:
	UF : 0, UT : 6,		CONFIG : 'N U T, 0, 0, 0',
	X =  487.295  mm,	Y =   -196.481  mm,	Z =   -263.764  mm,
	W =  90.000 deg,	P =   0.000 deg,	R =   90.000 deg
};
P[161]{
   GP1:
	UF : 0, UT : 6,		CONFIG : 'N U T, 0, 0, 0',
	X =  468.362  mm,	Y =   -207.462  mm,	Z =   -267.000  mm,
	W =  90.000 deg,	P =   0.000 deg,	R =   90.000 deg
};
P[162]{
   GP1:
	UF : 0, UT : 6,		CONFIG : 'N U T, 0, 0, 0',
	X =  426.797  mm,	Y =   -231.310  mm,	Z =   -267.000  mm,
	W =  90.000 deg,	P =   0.000 deg,	R =   90.000 deg
};
P[163]{
   GP1:
	UF : 0, UT : 6,		CONFIG : 'N U T, 0, 0, 0',
	X =  406.116  mm,	Y =   -243.329  mm,	Z =   -267.000  mm,
	W =  90.000 deg,	P =   0.000 deg,	R =   90.000 deg
};
P[164]{
   GP1:
	UF : 0, UT : 6,		CONFIG : 'N U T, 0, 0, 0',
	X =  385.124  mm,	Y =   -255.348  mm,	Z =   -267.000  mm,
	W =  90.000 deg,	P =   0.000 deg,	R =   90.000 deg
};
P[165]{
   GP1:
	UF : 0, UT : 6,		CONFIG : 'N U T, 0, 0, 0',
	X =  364.338  mm,	Y =   -267.372  mm,	Z =   -267.000  mm,
	W =  90.000 deg,	P =   0.000 deg,	R =   90.000 deg
};
P[166]{
   GP1:
	UF : 0, UT : 6,		CONFIG : 'N U T, 0, 0, 0',
	X =  322.888  mm,	Y =   -291.342  mm,	Z =   -267.000  mm,
	W =  90.000 deg,	P =   0.000 deg,	R =   90.000 deg
};
P[167]{
   GP1:
	UF : 0, UT : 6,		CONFIG : 'N U T, 0, 0, 0',
	X =  302.256  mm,	Y =   -303.386  mm,	Z =   -267.000  mm,
	W =  90.000 deg,	P =   0.000 deg,	R =   90.000 deg
};
P[168]{
   GP1:
	UF : 0, UT : 6,		CONFIG : 'N U T, 0, 0, 0',
	X =  281.269  mm,	Y =   -315.511  mm,	Z =   -267.000  mm,
	W =  90.000 deg,	P =   0.000 deg,	R =   90.000 deg
};
P[169]{
   GP1:
	UF : 0, UT : 6,		CONFIG : 'N U T, 0, 0, 0',
	X =  239.677  mm,	Y =   -339.423  mm,	Z =   -267.000  mm,
	W =  90.000 deg,	P =   0.000 deg,	R =   90.000 deg
};
P[170]{
   GP1:
	UF : 0, UT : 6,		CONFIG : 'N U T, 0, 0, 0',
	X =  198.097  mm,	Y =   -363.300  mm,	Z =   -267.000  mm,
	W =  90.000 deg,	P =   0.000 deg,	R =   90.000 deg
};
P[171]{
   GP1:
	UF : 0, UT : 6,		CONFIG : 'N U T, 0, 0, 0',
	X =  135.873  mm,	Y =   -399.405  mm,	Z =   -267.000  mm,
	W =  90.000 deg,	P =   0.000 deg,	R =   90.000 deg
};
P[172]{
   GP1:
	UF : 0, UT : 6,		CONFIG : 'N U T, 0, 0, 0',
	X =  115.069  mm,	Y =   -411.325  mm,	Z =   -267.000  mm,
	W =  90.000 deg,	P =   0.000 deg,	R =   90.000 deg
};
P[173]{
   GP1:
	UF : 0, UT : 6,		CONFIG : 'N U T, 0, 0, 0',
	X =  73.548  mm,	Y =   -435.396  mm,	Z =   -267.000  mm,
	W =  90.000 deg,	P =   0.000 deg,	R =   90.000 deg
};
P[174]{
   GP1:
	UF : 0, UT : 6,		CONFIG : 'N U T, 0, 0, 0',
	X =  -2.749  mm,	Y =   -479.250  mm,	Z =   -261.901  mm,
	W =  90.000 deg,	P =   0.000 deg,	R =   90.000 deg
};
P[175]{
   GP1:
	UF : 0, UT : 6,		CONFIG : 'N U T, 0, 0, 0',
	X =  -7.280  mm,	Y =   -482.139  mm,	Z =   -247.456  mm,
	W =  90.000 deg,	P =   0.000 deg,	R =   90.000 deg
};
P[176]{
   GP1:
	UF : 0, UT : 6,		CONFIG : 'N U T, 0, 0, 0',
	X =  11.339  mm,	Y =   -471.441  mm,	Z =   -267.000  mm,
	W =  90.000 deg,	P =   0.000 deg,	R =   90.000 deg
};
P[177]{
   GP1:
	UF : 0, UT : 6,		CONFIG : 'N U T, 0, 0, 0',
	X =  32.097  mm,	Y =   -459.529  mm,	Z =   -267.000  mm,
	W =  90.000 deg,	P =   0.000 deg,	R =   90.000 deg
};
P[178]{
   GP1:
	UF : 0, UT : 6,		CONFIG : 'N U T, 0, 0, 0',
	X =  52.866  mm,	Y =   -447.562  mm,	Z =   -267.000  mm,
	W =  90.000 deg,	P =   0.000 deg,	R =   90.000 deg
};
P[179]{
   GP1:
	UF : 0, UT : 6,		CONFIG : 'N U T, 0, 0, 0',
	X =  94.553  mm,	Y =   -423.385  mm,	Z =   -267.000  mm,
	W =  90.000 deg,	P =   0.000 deg,	R =   90.000 deg
};
P[180]{
   GP1:
	UF : 0, UT : 6,		CONFIG : 'N U T, 0, 0, 0',
	X =  156.891  mm,	Y =   -387.366  mm,	Z =   -267.000  mm,
	W =  90.000 deg,	P =   0.000 deg,	R =   90.000 deg
};
P[181]{
   GP1:
	UF : 0, UT : 6,		CONFIG : 'N U T, 0, 0, 0',
	X =  177.598  mm,	Y =   -375.508  mm,	Z =   -267.000  mm,
	W =  90.000 deg,	P =   0.000 deg,	R =   90.000 deg
};
P[182]{
   GP1:
	UF : 0, UT : 6,		CONFIG : 'N U T, 0, 0, 0',
	X =  218.982  mm,	Y =   -351.545  mm,	Z =   -267.000  mm,
	W =  90.000 deg,	P =   0.000 deg,	R =   90.000 deg
};
P[183]{
   GP1:
	UF : 0, UT : 6,		CONFIG : 'N U T, 0, 0, 0',
	X =  260.798  mm,	Y =   -327.631  mm,	Z =   -267.000  mm,
	W =  90.000 deg,	P =   0.000 deg,	R =   90.000 deg
};
P[184]{
   GP1:
	UF : 0, UT : 6,		CONFIG : 'N U T, 0, 0, 0',
	X =  343.689  mm,	Y =   -279.567  mm,	Z =   -267.000  mm,
	W =  90.000 deg,	P =   0.000 deg,	R =   90.000 deg
};
P[185]{
   GP1:
	UF : 0, UT : 6,		CONFIG : 'N U T, 0, 0, 0',
	X =  447.780  mm,	Y =   -219.561  mm,	Z =   -267.000  mm,
	W =  90.000 deg,	P =   0.000 deg,	R =   90.000 deg
};
P[186]{
   GP1:
	UF : 0, UT : 6,		CONFIG : 'N U T, 0, 0, 0',
	X =  506.643  mm,	Y =   -212.872  mm,	Z =   -247.497  mm,
	W =  90.000 deg,	P =   0.000 deg,	R =   90.000 deg
};
P[187]{
   GP1:
	UF : 0, UT : 6,		CONFIG : 'N U T, 0, 0, 0',
	X =  499.239  mm,	Y =   -217.240  mm,	Z =   -263.799  mm,
	W =  90.000 deg,	P =   0.000 deg,	R =   90.000 deg
};
P[188]{
   GP1:
	UF : 0, UT : 6,		CONFIG : 'N U T, 0, 0, 0',
	X =  418.106  mm,	Y =   -264.249  mm,	Z =   -267.000  mm,
	W =  90.000 deg,	P =   0.000 deg,	R =   90.000 deg
};
P[189]{
   GP1:
	UF : 0, UT : 6,		CONFIG : 'N U T, 0, 0, 0',
	X =  355.625  mm,	Y =   -300.059  mm,	Z =   -267.000  mm,
	W =  90.000 deg,	P =   0.000 deg,	R =   90.000 deg
};
P[190]{
   GP1:
	UF : 0, UT : 6,		CONFIG : 'N U T, 0, 0, 0',
	X =  334.959  mm,	Y =   -312.000  mm,	Z =   -267.000  mm,
	W =  90.000 deg,	P =   0.000 deg,	R =   90.000 deg
};
P[191]{
   GP1:
	UF : 0, UT : 6,		CONFIG : 'N U T, 0, 0, 0',
	X =  314.387  mm,	Y =   -324.119  mm,	Z =   -267.000  mm,
	W =  90.000 deg,	P =   0.000 deg,	R =   90.000 deg
};
P[192]{
   GP1:
	UF : 0, UT : 6,		CONFIG : 'N U T, 0, 0, 0',
	X =  293.577  mm,	Y =   -336.121  mm,	Z =   -267.000  mm,
	W =  90.000 deg,	P =   0.000 deg,	R =   90.000 deg
};
P[193]{
   GP1:
	UF : 0, UT : 6,		CONFIG : 'N U T, 0, 0, 0',
	X =  272.501  mm,	Y =   -347.946  mm,	Z =   -267.000  mm,
	W =  90.000 deg,	P =   0.000 deg,	R =   90.000 deg
};
P[194]{
   GP1:
	UF : 0, UT : 6,		CONFIG : 'N U T, 0, 0, 0',
	X =  251.705  mm,	Y =   -360.150  mm,	Z =   -267.000  mm,
	W =  90.000 deg,	P =   0.000 deg,	R =   90.000 deg
};
P[195]{
   GP1:
	UF : 0, UT : 6,		CONFIG : 'N U T, 0, 0, 0',
	X =  210.325  mm,	Y =   -384.203  mm,	Z =   -267.000  mm,
	W =  90.000 deg,	P =   0.000 deg,	R =   90.000 deg
};
P[196]{
   GP1:
	UF : 0, UT : 6,		CONFIG : 'N U T, 0, 0, 0',
	X =  189.409  mm,	Y =   -396.164  mm,	Z =   -267.000  mm,
	W =  90.000 deg,	P =   0.000 deg,	R =   90.000 deg
};
P[197]{
   GP1:
	UF : 0, UT : 6,		CONFIG : 'N U T, 0, 0, 0',
	X =  147.758  mm,	Y =   -420.142  mm,	Z =   -267.000  mm,
	W =  90.000 deg,	P =   0.000 deg,	R =   90.000 deg
};
P[198]{
   GP1:
	UF : 0, UT : 6,		CONFIG : 'N U T, 0, 0, 0',
	X =  106.222  mm,	Y =   -444.314  mm,	Z =   -267.000  mm,
	W =  90.000 deg,	P =   0.000 deg,	R =   90.000 deg
};
P[199]{
   GP1:
	UF : 0, UT : 6,		CONFIG : 'N U T, 0, 0, 0',
	X =  85.466  mm,	Y =   -456.298  mm,	Z =   -267.000  mm,
	W =  90.000 deg,	P =   0.000 deg,	R =   90.000 deg
};
P[200]{
   GP1:
	UF : 0, UT : 6,		CONFIG : 'N U T, 0, 0, 0',
	X =  44.109  mm,	Y =   -480.084  mm,	Z =   -267.000  mm,
	W =  90.000 deg,	P =   0.000 deg,	R =   90.000 deg
};
P[201]{
   GP1:
	UF : 0, UT : 6,		CONFIG : 'N U T, 0, 0, 0',
	X =  23.043  mm,	Y =   -492.313  mm,	Z =   -267.000  mm,
	W =  90.000 deg,	P =   0.000 deg,	R =   90.000 deg
};
P[202]{
   GP1:
	UF : 0, UT : 6,		CONFIG : 'N U T, 0, 0, 0',
	X =  9.172  mm,	Y =   -500.280  mm,	Z =   -261.504  mm,
	W =  90.000 deg,	P =   0.000 deg,	R =   90.000 deg
};
P[203]{
   GP1:
	UF : 0, UT : 6,		CONFIG : 'N U T, 0, 0, 0',
	X =  4.580  mm,	Y =   -502.838  mm,	Z =   -247.234  mm,
	W =  90.000 deg,	P =   0.000 deg,	R =   90.000 deg
};
P[204]{
   GP1:
	UF : 0, UT : 6,		CONFIG : 'N U T, 0, 0, 0',
	X =  64.858  mm,	Y =   -468.227  mm,	Z =   -267.000  mm,
	W =  90.000 deg,	P =   0.000 deg,	R =   90.000 deg
};
P[205]{
   GP1:
	UF : 0, UT : 6,		CONFIG : 'N U T, 0, 0, 0',
	X =  127.222  mm,	Y =   -432.250  mm,	Z =   -267.000  mm,
	W =  90.000 deg,	P =   0.000 deg,	R =   90.000 deg
};
P[206]{
   GP1:
	UF : 0, UT : 6,		CONFIG : 'N U T, 0, 0, 0',
	X =  168.741  mm,	Y =   -408.496  mm,	Z =   -267.000  mm,
	W =  90.000 deg,	P =   0.000 deg,	R =   90.000 deg
};
P[207]{
   GP1:
	UF : 0, UT : 6,		CONFIG : 'N U T, 0, 0, 0',
	X =  231.023  mm,	Y =   -372.334  mm,	Z =   -267.000  mm,
	W =  90.000 deg,	P =   0.000 deg,	R =   90.000 deg
};
P[208]{
   GP1:
	UF : 0, UT : 6,		CONFIG : 'N U T, 0, 0, 0',
	X =  376.725  mm,	Y =   -288.174  mm,	Z =   -267.000  mm,
	W =  90.000 deg,	P =   0.000 deg,	R =   90.000 deg
};
P[209]{
   GP1:
	UF : 0, UT : 6,		CONFIG : 'N U T, 0, 0, 0',
	X =  397.468  mm,	Y =   -276.234  mm,	Z =   -267.000  mm,
	W =  90.000 deg,	P =   0.000 deg,	R =   90.000 deg
};
P[210]{
   GP1:
	UF : 0, UT : 6,		CONFIG : 'N U T, 0, 0, 0',
	X =  438.932  mm,	Y =   -252.375  mm,	Z =   -267.000  mm,
	W =  90.000 deg,	P =   0.000 deg,	R =   90.000 deg
};
P[211]{
   GP1:
	UF : 0, UT : 6,		CONFIG : 'N U T, 0, 0, 0',
	X =  459.955  mm,	Y =   -240.522  mm,	Z =   -267.000  mm,
	W =  90.000 deg,	P =   0.000 deg,	R =   90.000 deg
};
P[212]{
   GP1:
	UF : 0, UT : 6,		CONFIG : 'N U T, 0, 0, 0',
	X =  480.593  mm,	Y =   -228.255  mm,	Z =   -267.000  mm,
	W =  90.000 deg,	P =   0.000 deg,	R =   90.000 deg
};
P[213]{
   GP1:
	UF : 0, UT : 6,		CONFIG : 'N U T, 0, 0, 0',
	X =  511.349  mm,	Y =   -238.004  mm,	Z =   -263.716  mm,
	W =  90.000 deg,	P =   0.000 deg,	R =   90.000 deg
};
P[214]{
   GP1:
	UF : 0, UT : 6,		CONFIG : 'N U T, 0, 0, 0',
	X =  492.432  mm,	Y =   -249.018  mm,	Z =   -267.000  mm,
	W =  90.000 deg,	P =   0.000 deg,	R =   90.000 deg
};
P[215]{
   GP1:
	UF : 0, UT : 6,		CONFIG : 'N U T, 0, 0, 0',
	X =  471.780  mm,	Y =   -260.975  mm,	Z =   -267.000  mm,
	W =  90.000 deg,	P =   0.000 deg,	R =   90.000 deg
};
P[216]{
   GP1:
	UF : 0, UT : 6,		CONFIG : 'N U T, 0, 0, 0',
	X =  430.050  mm,	Y =   -284.965  mm,	Z =   -267.000  mm,
	W =  90.000 deg,	P =   0.000 deg,	R =   90.000 deg
};
P[217]{
   GP1:
	UF : 0, UT : 6,		CONFIG : 'N U T, 0, 0, 0',
	X =  367.748  mm,	Y =   -320.901  mm,	Z =   -267.000  mm,
	W =  90.000 deg,	P =   0.000 deg,	R =   90.000 deg
};
P[218]{
   GP1:
	UF : 0, UT : 6,		CONFIG : 'N U T, 0, 0, 0',
	X =  346.983  mm,	Y =   -332.937  mm,	Z =   -267.000  mm,
	W =  90.000 deg,	P =   0.000 deg,	R =   90.000 deg
};
P[219]{
   GP1:
	UF : 0, UT : 6,		CONFIG : 'N U T, 0, 0, 0',
	X =  326.168  mm,	Y =   -344.857  mm,	Z =   -267.000  mm,
	W =  90.000 deg,	P =   0.000 deg,	R =   90.000 deg
};
P[220]{
   GP1:
	UF : 0, UT : 6,		CONFIG : 'N U T, 0, 0, 0',
	X =  305.520  mm,	Y =   -356.822  mm,	Z =   -267.000  mm,
	W =  90.000 deg,	P =   0.000 deg,	R =   90.000 deg
};
P[221]{
   GP1:
	UF : 0, UT : 6,		CONFIG : 'N U T, 0, 0, 0',
	X =  263.830  mm,	Y =   -380.936  mm,	Z =   -267.000  mm,
	W =  90.000 deg,	P =   0.000 deg,	R =   90.000 deg
};
P[222]{
   GP1:
	UF : 0, UT : 6,		CONFIG : 'N U T, 0, 0, 0',
	X =  242.945  mm,	Y =   -393.070  mm,	Z =   -267.000  mm,
	W =  90.000 deg,	P =   0.000 deg,	R =   90.000 deg
};
P[223]{
   GP1:
	UF : 0, UT : 6,		CONFIG : 'N U T, 0, 0, 0',
	X =  222.234  mm,	Y =   -404.921  mm,	Z =   -267.000  mm,
	W =  90.000 deg,	P =   0.000 deg,	R =   90.000 deg
};
P[224]{
   GP1:
	UF : 0, UT : 6,		CONFIG : 'N U T, 0, 0, 0',
	X =  201.509  mm,	Y =   -416.997  mm,	Z =   -267.000  mm,
	W =  90.000 deg,	P =   0.000 deg,	R =   90.000 deg
};
P[225]{
   GP1:
	UF : 0, UT : 6,		CONFIG : 'N U T, 0, 0, 0',
	X =  180.817  mm,	Y =   -428.965  mm,	Z =   -267.000  mm,
	W =  90.000 deg,	P =   0.000 deg,	R =   90.000 deg
};
P[226]{
   GP1:
	UF : 0, UT : 6,		CONFIG : 'N U T, 0, 0, 0',
	X =  118.291  mm,	Y =   -465.026  mm,	Z =   -267.000  mm,
	W =  90.000 deg,	P =   0.000 deg,	R =   90.000 deg
};
P[227]{
   GP1:
	UF : 0, UT : 6,		CONFIG : 'N U T, 0, 0, 0',
	X =  97.464  mm,	Y =   -476.829  mm,	Z =   -267.000  mm,
	W =  90.000 deg,	P =   0.000 deg,	R =   90.000 deg
};
P[228]{
   GP1:
	UF : 0, UT : 6,		CONFIG : 'N U T, 0, 0, 0',
	X =  76.838  mm,	Y =   -488.965  mm,	Z =   -267.000  mm,
	W =  90.000 deg,	P =   0.000 deg,	R =   90.000 deg
};
P[229]{
   GP1:
	UF : 0, UT : 6,		CONFIG : 'N U T, 0, 0, 0',
	X =  55.946  mm,	Y =   -501.022  mm,	Z =   -267.000  mm,
	W =  90.000 deg,	P =   0.000 deg,	R =   90.000 deg
};
P[230]{
   GP1:
	UF : 0, UT : 6,		CONFIG : 'N U T, 0, 0, 0',
	X =  21.362  mm,	Y =   -520.931  mm,	Z =   -261.929  mm,
	W =  90.000 deg,	P =   0.000 deg,	R =   90.000 deg
};
P[231]{
   GP1:
	UF : 0, UT : 6,		CONFIG : 'N U T, 0, 0, 0',
	X =  16.644  mm,	Y =   -523.588  mm,	Z =   -247.434  mm,
	W =  90.000 deg,	P =   0.000 deg,	R =   90.000 deg
};
P[232]{
   GP1:
	UF : 0, UT : 6,		CONFIG : 'N U T, 0, 0, 0',
	X =  35.280  mm,	Y =   -513.257  mm,	Z =   -267.000  mm,
	W =  90.000 deg,	P =   0.000 deg,	R =   90.000 deg
};
P[233]{
   GP1:
	UF : 0, UT : 6,		CONFIG : 'N U T, 0, 0, 0',
	X =  139.311  mm,	Y =   -452.957  mm,	Z =   -267.000  mm,
	W =  90.000 deg,	P =   0.000 deg,	R =   90.000 deg
};
P[234]{
   GP1:
	UF : 0, UT : 6,		CONFIG : 'N U T, 0, 0, 0',
	X =  160.019  mm,	Y =   -441.025  mm,	Z =   -267.000  mm,
	W =  90.000 deg,	P =   0.000 deg,	R =   90.000 deg
};
P[235]{
   GP1:
	UF : 0, UT : 6,		CONFIG : 'N U T, 0, 0, 0',
	X =  284.630  mm,	Y =   -369.149  mm,	Z =   -267.000  mm,
	W =  90.000 deg,	P =   0.000 deg,	R =   90.000 deg
};
P[236]{
   GP1:
	UF : 0, UT : 6,		CONFIG : 'N U T, 0, 0, 0',
	X =  388.465  mm,	Y =   -309.341  mm,	Z =   -267.000  mm,
	W =  90.000 deg,	P =   0.000 deg,	R =   90.000 deg
};
P[237]{
   GP1:
	UF : 0, UT : 6,		CONFIG : 'N U T, 0, 0, 0',
	X =  409.432  mm,	Y =   -297.071  mm,	Z =   -267.000  mm,
	W =  90.000 deg,	P =   0.000 deg,	R =   90.000 deg
};
P[238]{
   GP1:
	UF : 0, UT : 6,		CONFIG : 'N U T, 0, 0, 0',
	X =  450.796  mm,	Y =   -273.094  mm,	Z =   -267.000  mm,
	W =  90.000 deg,	P =   0.000 deg,	R =   90.000 deg
};
P[239]{
   GP1:
	UF : 0, UT : 6,		CONFIG : 'N U T, 0, 0, 0',
	X =  518.785  mm,	Y =   -233.872  mm,	Z =   -247.455  mm,
	W =  90.000 deg,	P =   0.000 deg,	R =   90.000 deg
};
P[240]{
   GP1:
	UF : 0, UT : 6,		CONFIG : 'N U T, 0, 0, 0',
	X =  523.378  mm,	Y =   -258.813  mm,	Z =   -263.746  mm,
	W =  90.000 deg,	P =   0.000 deg,	R =   90.000 deg
};
P[241]{
   GP1:
	UF : 0, UT : 6,		CONFIG : 'N U T, 0, 0, 0',
	X =  483.704  mm,	Y =   -281.715  mm,	Z =   -267.000  mm,
	W =  90.000 deg,	P =   0.000 deg,	R =   90.000 deg
};
P[242]{
   GP1:
	UF : 0, UT : 6,		CONFIG : 'N U T, 0, 0, 0',
	X =  441.943  mm,	Y =   -305.877  mm,	Z =   -267.000  mm,
	W =  90.000 deg,	P =   0.000 deg,	R =   90.000 deg
};
P[243]{
   GP1:
	UF : 0, UT : 6,		CONFIG : 'N U T, 0, 0, 0',
	X =  421.450  mm,	Y =   -317.554  mm,	Z =   -267.000  mm,
	W =  90.000 deg,	P =   0.000 deg,	R =   90.000 deg
};
P[244]{
   GP1:
	UF : 0, UT : 6,		CONFIG : 'N U T, 0, 0, 0',
	X =  359.066  mm,	Y =   -353.709  mm,	Z =   -267.000  mm,
	W =  90.000 deg,	P =   0.000 deg,	R =   90.000 deg
};
P[245]{
   GP1:
	UF : 0, UT : 6,		CONFIG : 'N U T, 0, 0, 0',
	X =  317.350  mm,	Y =   -377.733  mm,	Z =   -267.000  mm,
	W =  90.000 deg,	P =   0.000 deg,	R =   90.000 deg
};
P[246]{
   GP1:
	UF : 0, UT : 6,		CONFIG : 'N U T, 0, 0, 0',
	X =  296.407  mm,	Y =   -389.821  mm,	Z =   -267.000  mm,
	W =  90.000 deg,	P =   0.000 deg,	R =   90.000 deg
};
P[247]{
   GP1:
	UF : 0, UT : 6,		CONFIG : 'N U T, 0, 0, 0',
	X =  275.944  mm,	Y =   -401.651  mm,	Z =   -267.000  mm,
	W =  90.000 deg,	P =   0.000 deg,	R =   90.000 deg
};
P[248]{
   GP1:
	UF : 0, UT : 6,		CONFIG : 'N U T, 0, 0, 0',
	X =  192.869  mm,	Y =   -449.644  mm,	Z =   -267.000  mm,
	W =  90.000 deg,	P =   0.000 deg,	R =   90.000 deg
};
P[249]{
   GP1:
	UF : 0, UT : 6,		CONFIG : 'N U T, 0, 0, 0',
	X =  67.829  mm,	Y =   -521.738  mm,	Z =   -267.000  mm,
	W =  90.000 deg,	P =   0.000 deg,	R =   90.000 deg
};
P[250]{
   GP1:
	UF : 0, UT : 6,		CONFIG : 'N U T, 0, 0, 0',
	X =  47.352  mm,	Y =   -533.633  mm,	Z =   -267.000  mm,
	W =  90.000 deg,	P =   0.000 deg,	R =   90.000 deg
};
P[251]{
   GP1:
	UF : 0, UT : 6,		CONFIG : 'N U T, 0, 0, 0',
	X =  33.339  mm,	Y =   -541.745  mm,	Z =   -261.892  mm,
	W =  90.000 deg,	P =   0.000 deg,	R =   90.000 deg
};
P[252]{
   GP1:
	UF : 0, UT : 6,		CONFIG : 'N U T, 0, 0, 0',
	X =  28.755  mm,	Y =   -544.600  mm,	Z =   -247.383  mm,
	W =  90.000 deg,	P =   0.000 deg,	R =   90.000 deg
};
P[253]{
   GP1:
	UF : 0, UT : 6,		CONFIG : 'N U T, 0, 0, 0',
	X =  88.854  mm,	Y =   -509.995  mm,	Z =   -267.000  mm,
	W =  90.000 deg,	P =   0.000 deg,	R =   90.000 deg
};
P[254]{
   GP1:
	UF : 0, UT : 6,		CONFIG : 'N U T, 0, 0, 0',
	X =  109.644  mm,	Y =   -497.790  mm,	Z =   -267.000  mm,
	W =  90.000 deg,	P =   0.000 deg,	R =   90.000 deg
};
P[255]{
   GP1:
	UF : 0, UT : 6,		CONFIG : 'N U T, 0, 0, 0',
	X =  130.441  mm,	Y =   -485.888  mm,	Z =   -267.000  mm,
	W =  90.000 deg,	P =   0.000 deg,	R =   90.000 deg
};
P[256]{
   GP1:
	UF : 0, UT : 6,		CONFIG : 'N U T, 0, 0, 0',
	X =  151.393  mm,	Y =   -473.842  mm,	Z =   -267.000  mm,
	W =  90.000 deg,	P =   0.000 deg,	R =   90.000 deg
};
P[257]{
   GP1:
	UF : 0, UT : 6,		CONFIG : 'N U T, 0, 0, 0',
	X =  172.086  mm,	Y =   -461.775  mm,	Z =   -267.000  mm,
	W =  90.000 deg,	P =   0.000 deg,	R =   90.000 deg
};
P[258]{
   GP1:
	UF : 0, UT : 6,		CONFIG : 'N U T, 0, 0, 0',
	X =  213.475  mm,	Y =   -437.949  mm,	Z =   -267.000  mm,
	W =  90.000 deg,	P =   0.000 deg,	R =   90.000 deg
};
P[259]{
   GP1:
	UF : 0, UT : 6,		CONFIG : 'N U T, 0, 0, 0',
	X =  234.385  mm,	Y =   -425.995  mm,	Z =   -267.000  mm,
	W =  90.000 deg,	P =   0.000 deg,	R =   90.000 deg
};
P[260]{
   GP1:
	UF : 0, UT : 6,		CONFIG : 'N U T, 0, 0, 0',
	X =  255.078  mm,	Y =   -413.864  mm,	Z =   -267.000  mm,
	W =  90.000 deg,	P =   0.000 deg,	R =   90.000 deg
};
P[261]{
   GP1:
	UF : 0, UT : 6,		CONFIG : 'N U T, 0, 0, 0',
	X =  338.222  mm,	Y =   -365.960  mm,	Z =   -267.000  mm,
	W =  90.000 deg,	P =   0.000 deg,	R =   90.000 deg
};
P[262]{
   GP1:
	UF : 0, UT : 6,		CONFIG : 'N U T, 0, 0, 0',
	X =  379.917  mm,	Y =   -341.771  mm,	Z =   -267.000  mm,
	W =  90.000 deg,	P =   0.000 deg,	R =   90.000 deg
};
P[263]{
   GP1:
	UF : 0, UT : 6,		CONFIG : 'N U T, 0, 0, 0',
	X =  400.487  mm,	Y =   -329.885  mm,	Z =   -267.000  mm,
	W =  90.000 deg,	P =   0.000 deg,	R =   90.000 deg
};
P[264]{
   GP1:
	UF : 0, UT : 6,		CONFIG : 'N U T, 0, 0, 0',
	X =  463.081  mm,	Y =   -293.964  mm,	Z =   -267.000  mm,
	W =  90.000 deg,	P =   0.000 deg,	R =   90.000 deg
};
P[265]{
   GP1:
	UF : 0, UT : 6,		CONFIG : 'N U T, 0, 0, 0',
	X =  504.489  mm,	Y =   -269.882  mm,	Z =   -267.000  mm,
	W =  90.000 deg,	P =   0.000 deg,	R =   90.000 deg
};
P[266]{
   GP1:
	UF : 0, UT : 6,		CONFIG : 'N U T, 0, 0, 0',
	X =  530.840  mm,	Y =   -254.670  mm,	Z =   -247.344  mm,
	W =  90.000 deg,	P =   0.000 deg,	R =   90.000 deg
};
P[267]{
   GP1:
	UF : 0, UT : 6,		CONFIG : 'N U T, 0, 0, 0',
	X =  542.720  mm,	Y =   -275.316  mm,	Z =   -247.443  mm,
	W =  90.000 deg,	P =   0.000 deg,	R =   90.000 deg
};
P[268]{
   GP1:
	UF : 0, UT : 6,		CONFIG : 'N U T, 0, 0, 0',
	X =  535.290  mm,	Y =   -279.558  mm,	Z =   -263.769  mm,
	W =  90.000 deg,	P =   0.000 deg,	R =   90.000 deg
};
P[269]{
   GP1:
	UF : 0, UT : 6,		CONFIG : 'N U T, 0, 0, 0',
	X =  474.862  mm,	Y =   -314.467  mm,	Z =   -267.000  mm,
	W =  90.000 deg,	P =   0.000 deg,	R =   90.000 deg
};
P[270]{
   GP1:
	UF : 0, UT : 6,		CONFIG : 'N U T, 0, 0, 0',
	X =  453.954  mm,	Y =   -326.385  mm,	Z =   -267.000  mm,
	W =  90.000 deg,	P =   0.000 deg,	R =   90.000 deg
};
P[271]{
   GP1:
	UF : 0, UT : 6,		CONFIG : 'N U T, 0, 0, 0',
	X =  370.908  mm,	Y =   -374.464  mm,	Z =   -267.000  mm,
	W =  90.000 deg,	P =   0.000 deg,	R =   90.000 deg
};
P[272]{
   GP1:
	UF : 0, UT : 6,		CONFIG : 'N U T, 0, 0, 0',
	X =  350.065  mm,	Y =   -386.546  mm,	Z =   -267.000  mm,
	W =  90.000 deg,	P =   0.000 deg,	R =   90.000 deg
};
P[273]{
   GP1:
	UF : 0, UT : 6,		CONFIG : 'N U T, 0, 0, 0',
	X =  246.124  mm,	Y =   -446.617  mm,	Z =   -267.000  mm,
	W =  90.000 deg,	P =   0.000 deg,	R =   90.000 deg
};
P[274]{
   GP1:
	UF : 0, UT : 6,		CONFIG : 'N U T, 0, 0, 0',
	X =  225.505  mm,	Y =   -458.518  mm,	Z =   -267.000  mm,
	W =  90.000 deg,	P =   0.000 deg,	R =   90.000 deg
};
P[275]{
   GP1:
	UF : 0, UT : 6,		CONFIG : 'N U T, 0, 0, 0',
	X =  204.764  mm,	Y =   -470.534  mm,	Z =   -267.000  mm,
	W =  90.000 deg,	P =   0.000 deg,	R =   90.000 deg
};
P[276]{
   GP1:
	UF : 0, UT : 6,		CONFIG : 'N U T, 0, 0, 0',
	X =  183.956  mm,	Y =   -482.541  mm,	Z =   -267.000  mm,
	W =  90.000 deg,	P =   0.000 deg,	R =   90.000 deg
};
P[277]{
   GP1:
	UF : 0, UT : 6,		CONFIG : 'N U T, 0, 0, 0',
	X =  142.336  mm,	Y =   -506.597  mm,	Z =   -267.000  mm,
	W =  90.000 deg,	P =   0.000 deg,	R =   90.000 deg
};
P[278]{
   GP1:
	UF : 0, UT : 6,		CONFIG : 'N U T, 0, 0, 0',
	X =  100.703  mm,	Y =   -530.574  mm,	Z =   -267.000  mm,
	W =  90.000 deg,	P =   0.000 deg,	R =   90.000 deg
};
P[279]{
   GP1:
	UF : 0, UT : 6,		CONFIG : 'N U T, 0, 0, 0',
	X =  79.853  mm,	Y =   -542.532  mm,	Z =   -267.000  mm,
	W =  90.000 deg,	P =   0.000 deg,	R =   90.000 deg
};
P[280]{
   GP1:
	UF : 0, UT : 6,		CONFIG : 'N U T, 0, 0, 0',
	X =  59.361  mm,	Y =   -554.501  mm,	Z =   -267.000  mm,
	W =  90.000 deg,	P =   0.000 deg,	R =   90.000 deg
};
P[281]{
   GP1:
	UF : 0, UT : 6,		CONFIG : 'N U T, 0, 0, 0',
	X =  40.792  mm,	Y =   -565.419  mm,	Z =   -247.423  mm,
	W =  90.000 deg,	P =   0.000 deg,	R =   90.000 deg
};
P[282]{
   GP1:
	UF : 0, UT : 6,		CONFIG : 'N U T, 0, 0, 0',
	X =  45.429  mm,	Y =   -562.817  mm,	Z =   -261.759  mm,
	W =  90.000 deg,	P =   0.000 deg,	R =   90.000 deg
};
P[283]{
   GP1:
	UF : 0, UT : 6,		CONFIG : 'N U T, 0, 0, 0',
	X =  121.612  mm,	Y =   -518.618  mm,	Z =   -267.000  mm,
	W =  90.000 deg,	P =   0.000 deg,	R =   90.000 deg
};
P[284]{
   GP1:
	UF : 0, UT : 6,		CONFIG : 'N U T, 0, 0, 0',
	X =  163.206  mm,	Y =   -494.805  mm,	Z =   -267.000  mm,
	W =  90.000 deg,	P =   0.000 deg,	R =   90.000 deg
};
P[285]{
   GP1:
	UF : 0, UT : 6,		CONFIG : 'N U T, 0, 0, 0',
	X =  267.020  mm,	Y =   -434.732  mm,	Z =   -267.000  mm,
	W =  90.000 deg,	P =   0.000 deg,	R =   90.000 deg
};
P[286]{
   GP1:
	UF : 0, UT : 6,		CONFIG : 'N U T, 0, 0, 0',
	X =  287.936  mm,	Y =   -422.605  mm,	Z =   -267.000  mm,
	W =  90.000 deg,	P =   0.000 deg,	R =   90.000 deg
};
P[287]{
   GP1:
	UF : 0, UT : 6,		CONFIG : 'N U T, 0, 0, 0',
	X =  308.707  mm,	Y =   -410.761  mm,	Z =   -267.000  mm,
	W =  90.000 deg,	P =   0.000 deg,	R =   90.000 deg
};
P[288]{
   GP1:
	UF : 0, UT : 6,		CONFIG : 'N U T, 0, 0, 0',
	X =  329.599  mm,	Y =   -398.566  mm,	Z =   -267.000  mm,
	W =  90.000 deg,	P =   0.000 deg,	R =   90.000 deg
};
P[289]{
   GP1:
	UF : 0, UT : 6,		CONFIG : 'N U T, 0, 0, 0',
	X =  391.725  mm,	Y =   -362.842  mm,	Z =   -267.000  mm,
	W =  90.000 deg,	P =   0.000 deg,	R =   90.000 deg
};
P[290]{
   GP1:
	UF : 0, UT : 6,		CONFIG : 'N U T, 0, 0, 0',
	X =  412.656  mm,	Y =   -350.564  mm,	Z =   -267.000  mm,
	W =  90.000 deg,	P =   0.000 deg,	R =   90.000 deg
};
P[291]{
   GP1:
	UF : 0, UT : 6,		CONFIG : 'N U T, 0, 0, 0',
	X =  433.300  mm,	Y =   -338.675  mm,	Z =   -267.000  mm,
	W =  90.000 deg,	P =   0.000 deg,	R =   90.000 deg
};
P[292]{
   GP1:
	UF : 0, UT : 6,		CONFIG : 'N U T, 0, 0, 0',
	X =  495.657  mm,	Y =   -302.729  mm,	Z =   -267.000  mm,
	W =  90.000 deg,	P =   0.000 deg,	R =   90.000 deg
};
P[293]{
   GP1:
	UF : 0, UT : 6,		CONFIG : 'N U T, 0, 0, 0',
	X =  516.442  mm,	Y =   -290.818  mm,	Z =   -267.000  mm,
	W =  90.000 deg,	P =   0.000 deg,	R =   90.000 deg
};
P[294]{
   GP1:
	UF : 0, UT : 6,		CONFIG : 'N U T, 0, 0, 0',
	X =  547.245  mm,	Y =   -300.447  mm,	Z =   -263.824  mm,
	W =  90.000 deg,	P =   0.000 deg,	R =   90.000 deg
};
P[295]{
   GP1:
	UF : 0, UT : 6,		CONFIG : 'N U T, 0, 0, 0',
	X =  528.287  mm,	Y =   -311.166  mm,	Z =   -267.000  mm,
	W =  90.000 deg,	P =   0.000 deg,	R =   90.000 deg
};
P[296]{
   GP1:
	UF : 0, UT : 6,		CONFIG : 'N U T, 0, 0, 0',
	X =  486.904  mm,	Y =   -335.200  mm,	Z =   -267.000  mm,
	W =  90.000 deg,	P =   0.000 deg,	R =   90.000 deg
};
P[297]{
   GP1:
	UF : 0, UT : 6,		CONFIG : 'N U T, 0, 0, 0',
	X =  465.809  mm,	Y =   -347.405  mm,	Z =   -267.000  mm,
	W =  90.000 deg,	P =   0.000 deg,	R =   90.000 deg
};
P[298]{
   GP1:
	UF : 0, UT : 6,		CONFIG : 'N U T, 0, 0, 0',
	X =  445.086  mm,	Y =   -359.520  mm,	Z =   -267.000  mm,
	W =  90.000 deg,	P =   0.000 deg,	R =   90.000 deg
};
P[299]{
   GP1:
	UF : 0, UT : 6,		CONFIG : 'N U T, 0, 0, 0',
	X =  403.751  mm,	Y =   -383.331  mm,	Z =   -267.000  mm,
	W =  90.000 deg,	P =   0.000 deg,	R =   90.000 deg
};
P[300]{
   GP1:
	UF : 0, UT : 6,		CONFIG : 'N U T, 0, 0, 0',
	X =  362.215  mm,	Y =   -407.279  mm,	Z =   -267.000  mm,
	W =  90.000 deg,	P =   0.000 deg,	R =   90.000 deg
};
P[301]{
   GP1:
	UF : 0, UT : 6,		CONFIG : 'N U T, 0, 0, 0',
	X =  341.387  mm,	Y =   -419.311  mm,	Z =   -267.000  mm,
	W =  90.000 deg,	P =   0.000 deg,	R =   90.000 deg
};
P[302]{
   GP1:
	UF : 0, UT : 6,		CONFIG : 'N U T, 0, 0, 0',
	X =  320.401  mm,	Y =   -431.442  mm,	Z =   -267.000  mm,
	W =  90.000 deg,	P =   0.000 deg,	R =   90.000 deg
};
P[303]{
   GP1:
	UF : 0, UT : 6,		CONFIG : 'N U T, 0, 0, 0',
	X =  299.682  mm,	Y =   -443.418  mm,	Z =   -267.000  mm,
	W =  90.000 deg,	P =   0.000 deg,	R =   90.000 deg
};
P[304]{
   GP1:
	UF : 0, UT : 6,		CONFIG : 'N U T, 0, 0, 0',
	X =  279.062  mm,	Y =   -455.316  mm,	Z =   -267.000  mm,
	W =  90.000 deg,	P =   0.000 deg,	R =   90.000 deg
};
P[305]{
   GP1:
	UF : 0, UT : 6,		CONFIG : 'N U T, 0, 0, 0',
	X =  258.114  mm,	Y =   -467.293  mm,	Z =   -267.000  mm,
	W =  90.000 deg,	P =   0.000 deg,	R =   90.000 deg
};
P[306]{
   GP1:
	UF : 0, UT : 6,		CONFIG : 'N U T, 0, 0, 0',
	X =  237.705  mm,	Y =   -479.262  mm,	Z =   -267.000  mm,
	W =  90.000 deg,	P =   0.000 deg,	R =   90.000 deg
};
P[307]{
   GP1:
	UF : 0, UT : 6,		CONFIG : 'N U T, 0, 0, 0',
	X =  216.598  mm,	Y =   -491.277  mm,	Z =   -267.000  mm,
	W =  90.000 deg,	P =   0.000 deg,	R =   90.000 deg
};
P[308]{
   GP1:
	UF : 0, UT : 6,		CONFIG : 'N U T, 0, 0, 0',
	X =  195.905  mm,	Y =   -503.294  mm,	Z =   -267.000  mm,
	W =  90.000 deg,	P =   0.000 deg,	R =   90.000 deg
};
P[309]{
   GP1:
	UF : 0, UT : 6,		CONFIG : 'N U T, 0, 0, 0',
	X =  154.210  mm,	Y =   -527.393  mm,	Z =   -267.000  mm,
	W =  90.000 deg,	P =   0.000 deg,	R =   90.000 deg
};
P[310]{
   GP1:
	UF : 0, UT : 6,		CONFIG : 'N U T, 0, 0, 0',
	X =  133.520  mm,	Y =   -539.126  mm,	Z =   -267.000  mm,
	W =  90.000 deg,	P =   0.000 deg,	R =   90.000 deg
};
P[311]{
   GP1:
	UF : 0, UT : 6,		CONFIG : 'N U T, 0, 0, 0',
	X =  71.212  mm,	Y =   -575.113  mm,	Z =   -267.000  mm,
	W =  90.000 deg,	P =   0.000 deg,	R =   90.000 deg
};
P[312]{
   GP1:
	UF : 0, UT : 6,		CONFIG : 'N U T, 0, 0, 0',
	X =  52.692  mm,	Y =   -586.090  mm,	Z =   -247.339  mm,
	W =  90.000 deg,	P =   0.000 deg,	R =   90.000 deg
};
P[313]{
   GP1:
	UF : 0, UT : 6,		CONFIG : 'N U T, 0, 0, 0',
	X =  57.377  mm,	Y =   -583.437  mm,	Z =   -261.886  mm,
	W =  90.000 deg,	P =   0.000 deg,	R =   90.000 deg
};
P[314]{
   GP1:
	UF : 0, UT : 6,		CONFIG : 'N U T, 0, 0, 0',
	X =  92.028  mm,	Y =   -563.550  mm,	Z =   -267.000  mm,
	W =  90.000 deg,	P =   0.000 deg,	R =   90.000 deg
};
P[315]{
   GP1:
	UF : 0, UT : 6,		CONFIG : 'N U T, 0, 0, 0',
	X =  112.917  mm,	Y =   -551.512  mm,	Z =   -267.000  mm,
	W =  90.000 deg,	P =   0.000 deg,	R =   90.000 deg
};
P[316]{
   GP1:
	UF : 0, UT : 6,		CONFIG : 'N U T, 0, 0, 0',
	X =  175.320  mm,	Y =   -515.396  mm,	Z =   -267.000  mm,
	W =  90.000 deg,	P =   0.000 deg,	R =   90.000 deg
};
P[317]{
   GP1:
	UF : 0, UT : 6,		CONFIG : 'N U T, 0, 0, 0',
	X =  382.896  mm,	Y =   -395.523  mm,	Z =   -267.000  mm,
	W =  90.000 deg,	P =   0.000 deg,	R =   90.000 deg
};
P[318]{
   GP1:
	UF : 0, UT : 6,		CONFIG : 'N U T, 0, 0, 0',
	X =  424.458  mm,	Y =   -371.581  mm,	Z =   -267.000  mm,
	W =  90.000 deg,	P =   0.000 deg,	R =   90.000 deg
};
P[319]{
   GP1:
	UF : 0, UT : 6,		CONFIG : 'N U T, 0, 0, 0',
	X =  507.746  mm,	Y =   -323.548  mm,	Z =   -267.000  mm,
	W =  90.000 deg,	P =   0.000 deg,	R =   90.000 deg
};
P[320]{
   GP1:
	UF : 0, UT : 6,		CONFIG : 'N U T, 0, 0, 0',
	X =  554.836  mm,	Y =   -296.327  mm,	Z =   -247.482  mm,
	W =  90.000 deg,	P =   0.000 deg,	R =   90.000 deg
};
P[321]{
   GP1:
	UF : 0, UT : 6,		CONFIG : 'N U T, 0, 0, 0',
	X =  559.304  mm,	Y =   -321.202  mm,	Z =   -263.803  mm,
	W =  90.000 deg,	P =   0.000 deg,	R =   90.000 deg
};
P[322]{
   GP1:
	UF : 0, UT : 6,		CONFIG : 'N U T, 0, 0, 0',
	X =  540.278  mm,	Y =   -332.277  mm,	Z =   -267.000  mm,
	W =  90.000 deg,	P =   0.000 deg,	R =   90.000 deg
};
P[323]{
   GP1:
	UF : 0, UT : 6,		CONFIG : 'N U T, 0, 0, 0',
	X =  477.974  mm,	Y =   -368.146  mm,	Z =   -267.000  mm,
	W =  90.000 deg,	P =   0.000 deg,	R =   90.000 deg
};
P[324]{
   GP1:
	UF : 0, UT : 6,		CONFIG : 'N U T, 0, 0, 0',
	X =  394.817  mm,	Y =   -416.209  mm,	Z =   -267.000  mm,
	W =  90.000 deg,	P =   0.000 deg,	R =   90.000 deg
};
P[325]{
   GP1:
	UF : 0, UT : 6,		CONFIG : 'N U T, 0, 0, 0',
	X =  332.591  mm,	Y =   -452.117  mm,	Z =   -267.000  mm,
	W =  90.000 deg,	P =   0.000 deg,	R =   90.000 deg
};
P[326]{
   GP1:
	UF : 0, UT : 6,		CONFIG : 'N U T, 0, 0, 0',
	X =  290.913  mm,	Y =   -476.208  mm,	Z =   -267.000  mm,
	W =  90.000 deg,	P =   0.000 deg,	R =   90.000 deg
};
P[327]{
   GP1:
	UF : 0, UT : 6,		CONFIG : 'N U T, 0, 0, 0',
	X =  270.176  mm,	Y =   -488.138  mm,	Z =   -267.000  mm,
	W =  90.000 deg,	P =   0.000 deg,	R =   90.000 deg
};
P[328]{
   GP1:
	UF : 0, UT : 6,		CONFIG : 'N U T, 0, 0, 0',
	X =  228.578  mm,	Y =   -512.246  mm,	Z =   -267.000  mm,
	W =  90.000 deg,	P =   0.000 deg,	R =   90.000 deg
};
P[329]{
   GP1:
	UF : 0, UT : 6,		CONFIG : 'N U T, 0, 0, 0',
	X =  207.894  mm,	Y =   -524.188  mm,	Z =   -267.000  mm,
	W =  90.000 deg,	P =   0.000 deg,	R =   90.000 deg
};
P[330]{
   GP1:
	UF : 0, UT : 6,		CONFIG : 'N U T, 0, 0, 0',
	X =  187.158  mm,	Y =   -536.075  mm,	Z =   -267.000  mm,
	W =  90.000 deg,	P =   0.000 deg,	R =   90.000 deg
};
P[331]{
   GP1:
	UF : 0, UT : 6,		CONFIG : 'N U T, 0, 0, 0',
	X =  145.570  mm,	Y =   -559.925  mm,	Z =   -267.000  mm,
	W =  90.000 deg,	P =   0.000 deg,	R =   90.000 deg
};
P[332]{
   GP1:
	UF : 0, UT : 6,		CONFIG : 'N U T, 0, 0, 0',
	X =  103.939  mm,	Y =   -584.039  mm,	Z =   -267.000  mm,
	W =  90.000 deg,	P =   0.000 deg,	R =   90.000 deg
};
P[333]{
   GP1:
	UF : 0, UT : 6,		CONFIG : 'N U T, 0, 0, 0',
	X =  83.112  mm,	Y =   -596.084  mm,	Z =   -267.000  mm,
	W =  90.000 deg,	P =   0.000 deg,	R =   90.000 deg
};
P[334]{
   GP1:
	UF : 0, UT : 6,		CONFIG : 'N U T, 0, 0, 0',
	X =  64.609  mm,	Y =   -606.653  mm,	Z =   -247.444  mm,
	W =  90.000 deg,	P =   0.000 deg,	R =   90.000 deg
};
P[335]{
   GP1:
	UF : 0, UT : 6,		CONFIG : 'N U T, 0, 0, 0',
	X =  69.385  mm,	Y =   -604.172  mm,	Z =   -261.877  mm,
	W =  90.000 deg,	P =   0.000 deg,	R =   90.000 deg
};
P[336]{
   GP1:
	UF : 0, UT : 6,		CONFIG : 'N U T, 0, 0, 0',
	X =  124.733  mm,	Y =   -572.320  mm,	Z =   -267.000  mm,
	W =  90.000 deg,	P =   0.000 deg,	R =   90.000 deg
};
P[337]{
   GP1:
	UF : 0, UT : 6,		CONFIG : 'N U T, 0, 0, 0',
	X =  166.480  mm,	Y =   -548.196  mm,	Z =   -267.000  mm,
	W =  90.000 deg,	P =   0.000 deg,	R =   90.000 deg
};
P[338]{
   GP1:
	UF : 0, UT : 6,		CONFIG : 'N U T, 0, 0, 0',
	X =  249.621  mm,	Y =   -500.344  mm,	Z =   -267.000  mm,
	W =  90.000 deg,	P =   0.000 deg,	R =   90.000 deg
};
P[339]{
   GP1:
	UF : 0, UT : 6,		CONFIG : 'N U T, 0, 0, 0',
	X =  311.772  mm,	Y =   -464.265  mm,	Z =   -267.000  mm,
	W =  90.000 deg,	P =   0.000 deg,	R =   90.000 deg
};
P[340]{
   GP1:
	UF : 0, UT : 6,		CONFIG : 'N U T, 0, 0, 0',
	X =  353.397  mm,	Y =   -440.395  mm,	Z =   -267.000  mm,
	W =  90.000 deg,	P =   0.000 deg,	R =   90.000 deg
};
P[341]{
   GP1:
	UF : 0, UT : 6,		CONFIG : 'N U T, 0, 0, 0',
	X =  374.196  mm,	Y =   -428.228  mm,	Z =   -267.000  mm,
	W =  90.000 deg,	P =   0.000 deg,	R =   90.000 deg
};
P[342]{
   GP1:
	UF : 0, UT : 6,		CONFIG : 'N U T, 0, 0, 0',
	X =  415.929  mm,	Y =   -404.259  mm,	Z =   -267.000  mm,
	W =  90.000 deg,	P =   0.000 deg,	R =   90.000 deg
};
P[343]{
   GP1:
	UF : 0, UT : 6,		CONFIG : 'N U T, 0, 0, 0',
	X =  436.539  mm,	Y =   -392.369  mm,	Z =   -267.000  mm,
	W =  90.000 deg,	P =   0.000 deg,	R =   90.000 deg
};
P[344]{
   GP1:
	UF : 0, UT : 6,		CONFIG : 'N U T, 0, 0, 0',
	X =  457.289  mm,	Y =   -380.340  mm,	Z =   -267.000  mm,
	W =  90.000 deg,	P =   0.000 deg,	R =   90.000 deg
};
P[345]{
   GP1:
	UF : 0, UT : 6,		CONFIG : 'N U T, 0, 0, 0',
	X =  498.980  mm,	Y =   -356.143  mm,	Z =   -267.000  mm,
	W =  90.000 deg,	P =   0.000 deg,	R =   90.000 deg
};
P[346]{
   GP1:
	UF : 0, UT : 6,		CONFIG : 'N U T, 0, 0, 0',
	X =  519.504  mm,	Y =   -344.374  mm,	Z =   -267.000  mm,
	W =  90.000 deg,	P =   0.000 deg,	R =   90.000 deg
};
P[347]{
   GP1:
	UF : 0, UT : 6,		CONFIG : 'N U T, 0, 0, 0',
	X =  566.800  mm,	Y =   -316.983  mm,	Z =   -247.389  mm,
	W =  90.000 deg,	P =   0.000 deg,	R =   90.000 deg
};
P[348]{
   GP1:
	UF : 0, UT : 6,		CONFIG : 'N U T, 0, 0, 0',
	X =  571.399  mm,	Y =   -341.883  mm,	Z =   -263.779  mm,
	W =  90.000 deg,	P =   0.000 deg,	R =   90.000 deg
};
P[349]{
   GP1:
	UF : 0, UT : 6,		CONFIG : 'N U T, 0, 0, 0',
	X =  552.585  mm,	Y =   -352.768  mm,	Z =   -267.000  mm,
	W =  90.000 deg,	P =   0.000 deg,	R =   90.000 deg
};
P[350]{
   GP1:
	UF : 0, UT : 6,		CONFIG : 'N U T, 0, 0, 0',
	X =  510.899  mm,	Y =   -376.777  mm,	Z =   -267.000  mm,
	W =  90.000 deg,	P =   0.000 deg,	R =   90.000 deg
};
P[351]{
   GP1:
	UF : 0, UT : 6,		CONFIG : 'N U T, 0, 0, 0',
	X =  490.141  mm,	Y =   -388.808  mm,	Z =   -267.000  mm,
	W =  90.000 deg,	P =   0.000 deg,	R =   90.000 deg
};
P[352]{
   GP1:
	UF : 0, UT : 6,		CONFIG : 'N U T, 0, 0, 0',
	X =  469.401  mm,	Y =   -400.862  mm,	Z =   -267.000  mm,
	W =  90.000 deg,	P =   0.000 deg,	R =   90.000 deg
};
P[353]{
   GP1:
	UF : 0, UT : 6,		CONFIG : 'N U T, 0, 0, 0',
	X =  448.687  mm,	Y =   -412.877  mm,	Z =   -267.000  mm,
	W =  90.000 deg,	P =   0.000 deg,	R =   90.000 deg
};
P[354]{
   GP1:
	UF : 0, UT : 6,		CONFIG : 'N U T, 0, 0, 0',
	X =  427.661  mm,	Y =   -425.016  mm,	Z =   -267.000  mm,
	W =  90.000 deg,	P =   0.000 deg,	R =   90.000 deg
};
P[355]{
   GP1:
	UF : 0, UT : 6,		CONFIG : 'N U T, 0, 0, 0',
	X =  406.948  mm,	Y =   -436.874  mm,	Z =   -267.000  mm,
	W =  90.000 deg,	P =   0.000 deg,	R =   90.000 deg
};
P[356]{
   GP1:
	UF : 0, UT : 6,		CONFIG : 'N U T, 0, 0, 0',
	X =  365.529  mm,	Y =   -460.838  mm,	Z =   -267.000  mm,
	W =  90.000 deg,	P =   0.000 deg,	R =   90.000 deg
};
P[357]{
   GP1:
	UF : 0, UT : 6,		CONFIG : 'N U T, 0, 0, 0',
	X =  344.750  mm,	Y =   -472.859  mm,	Z =   -267.000  mm,
	W =  90.000 deg,	P =   0.000 deg,	R =   90.000 deg
};
P[358]{
   GP1:
	UF : 0, UT : 6,		CONFIG : 'N U T, 0, 0, 0',
	X =  303.029  mm,	Y =   -496.949  mm,	Z =   -267.000  mm,
	W =  90.000 deg,	P =   0.000 deg,	R =   90.000 deg
};
P[359]{
   GP1:
	UF : 0, UT : 6,		CONFIG : 'N U T, 0, 0, 0',
	X =  240.553  mm,	Y =   -532.970  mm,	Z =   -267.000  mm,
	W =  90.000 deg,	P =   0.000 deg,	R =   90.000 deg
};
P[360]{
   GP1:
	UF : 0, UT : 6,		CONFIG : 'N U T, 0, 0, 0',
	X =  220.018  mm,	Y =   -544.809  mm,	Z =   -267.000  mm,
	W =  90.000 deg,	P =   0.000 deg,	R =   90.000 deg
};
P[361]{
   GP1:
	UF : 0, UT : 6,		CONFIG : 'N U T, 0, 0, 0',
	X =  199.002  mm,	Y =   -556.796  mm,	Z =   -267.000  mm,
	W =  90.000 deg,	P =   0.000 deg,	R =   90.000 deg
};
P[362]{
   GP1:
	UF : 0, UT : 6,		CONFIG : 'N U T, 0, 0, 0',
	X =  115.838  mm,	Y =   -604.834  mm,	Z =   -267.000  mm,
	W =  90.000 deg,	P =   0.000 deg,	R =   90.000 deg
};
P[363]{
   GP1:
	UF : 0, UT : 6,		CONFIG : 'N U T, 0, 0, 0',
	X =  95.186  mm,	Y =   -616.850  mm,	Z =   -267.000  mm,
	W =  90.000 deg,	P =   0.000 deg,	R =   90.000 deg
};
P[364]{
   GP1:
	UF : 0, UT : 6,		CONFIG : 'N U T, 0, 0, 0',
	X =  76.761  mm,	Y =   -627.655  mm,	Z =   -247.508  mm,
	W =  90.000 deg,	P =   0.000 deg,	R =   90.000 deg
};
P[365]{
   GP1:
	UF : 0, UT : 6,		CONFIG : 'N U T, 0, 0, 0',
	X =  81.406  mm,	Y =   -625.034  mm,	Z =   -261.836  mm,
	W =  90.000 deg,	P =   0.000 deg,	R =   90.000 deg
};
P[366]{
   GP1:
	UF : 0, UT : 6,		CONFIG : 'N U T, 0, 0, 0',
	X =  137.005  mm,	Y =   -592.902  mm,	Z =   -267.000  mm,
	W =  90.000 deg,	P =   0.000 deg,	R =   90.000 deg
};
P[367]{
   GP1:
	UF : 0, UT : 6,		CONFIG : 'N U T, 0, 0, 0',
	X =  157.536  mm,	Y =   -581.155  mm,	Z =   -267.000  mm,
	W =  90.000 deg,	P =   0.000 deg,	R =   90.000 deg
};
P[368]{
   GP1:
	UF : 0, UT : 6,		CONFIG : 'N U T, 0, 0, 0',
	X =  178.231  mm,	Y =   -569.047  mm,	Z =   -267.000  mm,
	W =  90.000 deg,	P =   0.000 deg,	R =   90.000 deg
};
P[369]{
   GP1:
	UF : 0, UT : 6,		CONFIG : 'N U T, 0, 0, 0',
	X =  261.499  mm,	Y =   -521.017  mm,	Z =   -267.000  mm,
	W =  90.000 deg,	P =   0.000 deg,	R =   90.000 deg
};
P[370]{
   GP1:
	UF : 0, UT : 6,		CONFIG : 'N U T, 0, 0, 0',
	X =  282.162  mm,	Y =   -509.045  mm,	Z =   -267.000  mm,
	W =  90.000 deg,	P =   0.000 deg,	R =   90.000 deg
};
P[371]{
   GP1:
	UF : 0, UT : 6,		CONFIG : 'N U T, 0, 0, 0',
	X =  324.113  mm,	Y =   -484.984  mm,	Z =   -267.000  mm,
	W =  90.000 deg,	P =   0.000 deg,	R =   90.000 deg
};
P[372]{
   GP1:
	UF : 0, UT : 6,		CONFIG : 'N U T, 0, 0, 0',
	X =  386.122  mm,	Y =   -449.023  mm,	Z =   -267.000  mm,
	W =  90.000 deg,	P =   0.000 deg,	R =   90.000 deg
};
P[373]{
   GP1:
	UF : 0, UT : 6,		CONFIG : 'N U T, 0, 0, 0',
	X =  531.729  mm,	Y =   -364.993  mm,	Z =   -267.000  mm,
	W =  90.000 deg,	P =   0.000 deg,	R =   90.000 deg
};
P[374]{
   GP1:
	UF : 0, UT : 6,		CONFIG : 'N U T, 0, 0, 0',
	X =  578.894  mm,	Y =   -337.940  mm,	Z =   -247.405  mm,
	W =  90.000 deg,	P =   0.000 deg,	R =   90.000 deg
};
P[375]{
   GP1:
	UF : 0, UT : 6,		CONFIG : 'N U T, 0, 0, 0',
	X =  583.276  mm,	Y =   -362.724  mm,	Z =   -263.839  mm,
	W =  90.000 deg,	P =   0.000 deg,	R =   90.000 deg
};
P[376]{
   GP1:
	UF : 0, UT : 6,		CONFIG : 'N U T, 0, 0, 0',
	X =  523.061  mm,	Y =   -397.498  mm,	Z =   -267.000  mm,
	W =  90.000 deg,	P =   0.000 deg,	R =   90.000 deg
};
P[377]{
   GP1:
	UF : 0, UT : 6,		CONFIG : 'N U T, 0, 0, 0',
	X =  460.475  mm,	Y =   -433.759  mm,	Z =   -267.000  mm,
	W =  90.000 deg,	P =   0.000 deg,	R =   90.000 deg
};
P[378]{
   GP1:
	UF : 0, UT : 6,		CONFIG : 'N U T, 0, 0, 0',
	X =  398.100  mm,	Y =   -469.591  mm,	Z =   -267.000  mm,
	W =  90.000 deg,	P =   0.000 deg,	R =   90.000 deg
};
P[379]{
   GP1:
	UF : 0, UT : 6,		CONFIG : 'N U T, 0, 0, 0',
	X =  356.489  mm,	Y =   -493.771  mm,	Z =   -267.000  mm,
	W =  90.000 deg,	P =   0.000 deg,	R =   90.000 deg
};
P[380]{
   GP1:
	UF : 0, UT : 6,		CONFIG : 'N U T, 0, 0, 0',
	X =  335.935  mm,	Y =   -505.673  mm,	Z =   -267.000  mm,
	W =  90.000 deg,	P =   0.000 deg,	R =   90.000 deg
};
P[381]{
   GP1:
	UF : 0, UT : 6,		CONFIG : 'N U T, 0, 0, 0',
	X =  315.082  mm,	Y =   -517.702  mm,	Z =   -267.000  mm,
	W =  90.000 deg,	P =   0.000 deg,	R =   90.000 deg
};
P[382]{
   GP1:
	UF : 0, UT : 6,		CONFIG : 'N U T, 0, 0, 0',
	X =  294.346  mm,	Y =   -529.577  mm,	Z =   -267.000  mm,
	W =  90.000 deg,	P =   0.000 deg,	R =   90.000 deg
};
P[383]{
   GP1:
	UF : 0, UT : 6,		CONFIG : 'N U T, 0, 0, 0',
	X =  231.811  mm,	Y =   -565.729  mm,	Z =   -267.000  mm,
	W =  90.000 deg,	P =   0.000 deg,	R =   90.000 deg
};
P[384]{
   GP1:
	UF : 0, UT : 6,		CONFIG : 'N U T, 0, 0, 0',
	X =  211.188  mm,	Y =   -577.563  mm,	Z =   -267.000  mm,
	W =  90.000 deg,	P =   0.000 deg,	R =   90.000 deg
};
P[385]{
   GP1:
	UF : 0, UT : 6,		CONFIG : 'N U T, 0, 0, 0',
	X =  169.623  mm,	Y =   -601.695  mm,	Z =   -267.000  mm,
	W =  90.000 deg,	P =   0.000 deg,	R =   90.000 deg
};
P[386]{
   GP1:
	UF : 0, UT : 6,		CONFIG : 'N U T, 0, 0, 0',
	X =  148.981  mm,	Y =   -613.457  mm,	Z =   -267.000  mm,
	W =  90.000 deg,	P =   0.000 deg,	R =   90.000 deg
};
P[387]{
   GP1:
	UF : 0, UT : 6,		CONFIG : 'N U T, 0, 0, 0',
	X =  128.005  mm,	Y =   -625.709  mm,	Z =   -267.000  mm,
	W =  90.000 deg,	P =   0.000 deg,	R =   90.000 deg
};
P[388]{
   GP1:
	UF : 0, UT : 6,		CONFIG : 'N U T, 0, 0, 0',
	X =  107.283  mm,	Y =   -637.687  mm,	Z =   -267.000  mm,
	W =  90.000 deg,	P =   0.000 deg,	R =   90.000 deg
};
P[389]{
   GP1:
	UF : 0, UT : 6,		CONFIG : 'N U T, 0, 0, 0',
	X =  93.291  mm,	Y =   -645.613  mm,	Z =   -261.838  mm,
	W =  90.000 deg,	P =   0.000 deg,	R =   90.000 deg
};
P[390]{
   GP1:
	UF : 0, UT : 6,		CONFIG : 'N U T, 0, 0, 0',
	X =  88.692  mm,	Y =   -648.407  mm,	Z =   -247.384  mm,
	W =  90.000 deg,	P =   0.000 deg,	R =   90.000 deg
};
P[391]{
   GP1:
	UF : 0, UT : 6,		CONFIG : 'N U T, 0, 0, 0',
	X =  190.409  mm,	Y =   -589.806  mm,	Z =   -267.000  mm,
	W =  90.000 deg,	P =   0.000 deg,	R =   90.000 deg
};
P[392]{
   GP1:
	UF : 0, UT : 6,		CONFIG : 'N U T, 0, 0, 0',
	X =  252.752  mm,	Y =   -553.811  mm,	Z =   -267.000  mm,
	W =  90.000 deg,	P =   0.000 deg,	R =   90.000 deg
};
P[393]{
   GP1:
	UF : 0, UT : 6,		CONFIG : 'N U T, 0, 0, 0',
	X =  273.598  mm,	Y =   -541.789  mm,	Z =   -267.000  mm,
	W =  90.000 deg,	P =   0.000 deg,	R =   90.000 deg
};
P[394]{
   GP1:
	UF : 0, UT : 6,		CONFIG : 'N U T, 0, 0, 0',
	X =  377.408  mm,	Y =   -481.763  mm,	Z =   -267.000  mm,
	W =  90.000 deg,	P =   0.000 deg,	R =   90.000 deg
};
P[395]{
   GP1:
	UF : 0, UT : 6,		CONFIG : 'N U T, 0, 0, 0',
	X =  419.123  mm,	Y =   -457.815  mm,	Z =   -267.000  mm,
	W =  90.000 deg,	P =   0.000 deg,	R =   90.000 deg
};
P[396]{
   GP1:
	UF : 0, UT : 6,		CONFIG : 'N U T, 0, 0, 0',
	X =  439.892  mm,	Y =   -445.927  mm,	Z =   -267.000  mm,
	W =  90.000 deg,	P =   0.000 deg,	R =   90.000 deg
};
P[397]{
   GP1:
	UF : 0, UT : 6,		CONFIG : 'N U T, 0, 0, 0',
	X =  481.447  mm,	Y =   -421.691  mm,	Z =   -267.000  mm,
	W =  90.000 deg,	P =   0.000 deg,	R =   90.000 deg
};
P[398]{
   GP1:
	UF : 0, UT : 6,		CONFIG : 'N U T, 0, 0, 0',
	X =  502.005  mm,	Y =   -409.995  mm,	Z =   -267.000  mm,
	W =  90.000 deg,	P =   0.000 deg,	R =   90.000 deg
};
P[399]{
   GP1:
	UF : 0, UT : 6,		CONFIG : 'N U T, 0, 0, 0',
	X =  543.738  mm,	Y =   -385.778  mm,	Z =   -267.000  mm,
	W =  90.000 deg,	P =   0.000 deg,	R =   90.000 deg
};
P[400]{
   GP1:
	UF : 0, UT : 6,		CONFIG : 'N U T, 0, 0, 0',
	X =  564.423  mm,	Y =   -373.838  mm,	Z =   -267.000  mm,
	W =  90.000 deg,	P =   0.000 deg,	R =   90.000 deg
};
P[401]{
   GP1:
	UF : 0, UT : 6,		CONFIG : 'N U T, 0, 0, 0',
	X =  590.840  mm,	Y =   -358.624  mm,	Z =   -247.398  mm,
	W =  90.000 deg,	P =   0.000 deg,	R =   90.000 deg
};
P[402]{
   GP1:
	UF : 0, UT : 6,		CONFIG : 'N U T, 0, 0, 0',
	X =  576.281  mm,	Y =   -394.556  mm,	Z =   -267.000  mm,
	W =  90.000 deg,	P =   0.000 deg,	R =   90.000 deg
};
P[403]{
   GP1:
	UF : 0, UT : 6,		CONFIG : 'N U T, 0, 0, 0',
	X =  555.713  mm,	Y =   -406.314  mm,	Z =   -267.000  mm,
	W =  90.000 deg,	P =   0.000 deg,	R =   90.000 deg
};
P[404]{
   GP1:
	UF : 0, UT : 6,		CONFIG : 'N U T, 0, 0, 0',
	X =  534.884  mm,	Y =   -418.352  mm,	Z =   -267.000  mm,
	W =  90.000 deg,	P =   0.000 deg,	R =   90.000 deg
};
P[405]{
   GP1:
	UF : 0, UT : 6,		CONFIG : 'N U T, 0, 0, 0',
	X =  493.243  mm,	Y =   -442.297  mm,	Z =   -267.000  mm,
	W =  90.000 deg,	P =   0.000 deg,	R =   90.000 deg
};
P[406]{
   GP1:
	UF : 0, UT : 6,		CONFIG : 'N U T, 0, 0, 0',
	X =  410.370  mm,	Y =   -490.412  mm,	Z =   -267.000  mm,
	W =  90.000 deg,	P =   0.000 deg,	R =   90.000 deg
};
P[407]{
   GP1:
	UF : 0, UT : 6,		CONFIG : 'N U T, 0, 0, 0',
	X =  389.553  mm,	Y =   -502.335  mm,	Z =   -267.000  mm,
	W =  90.000 deg,	P =   0.000 deg,	R =   90.000 deg
};
P[408]{
   GP1:
	UF : 0, UT : 6,		CONFIG : 'N U T, 0, 0, 0',
	X =  306.113  mm,	Y =   -550.488  mm,	Z =   -267.000  mm,
	W =  90.000 deg,	P =   0.000 deg,	R =   90.000 deg
};
P[409]{
   GP1:
	UF : 0, UT : 6,		CONFIG : 'N U T, 0, 0, 0',
	X =  264.618  mm,	Y =   -574.509  mm,	Z =   -267.000  mm,
	W =  90.000 deg,	P =   0.000 deg,	R =   90.000 deg
};
P[410]{
   GP1:
	UF : 0, UT : 6,		CONFIG : 'N U T, 0, 0, 0',
	X =  243.651  mm,	Y =   -586.373  mm,	Z =   -267.000  mm,
	W =  90.000 deg,	P =   0.000 deg,	R =   90.000 deg
};
P[411]{
   GP1:
	UF : 0, UT : 6,		CONFIG : 'N U T, 0, 0, 0',
	X =  222.947  mm,	Y =   -598.419  mm,	Z =   -267.000  mm,
	W =  90.000 deg,	P =   0.000 deg,	R =   90.000 deg
};
P[412]{
   GP1:
	UF : 0, UT : 6,		CONFIG : 'N U T, 0, 0, 0',
	X =  160.629  mm,	Y =   -634.525  mm,	Z =   -267.000  mm,
	W =  90.000 deg,	P =   0.000 deg,	R =   90.000 deg
};
P[413]{
   GP1:
	UF : 0, UT : 6,		CONFIG : 'N U T, 0, 0, 0',
	X =  139.910  mm,	Y =   -646.475  mm,	Z =   -267.000  mm,
	W =  90.000 deg,	P =   0.000 deg,	R =   90.000 deg
};
P[414]{
   GP1:
	UF : 0, UT : 6,		CONFIG : 'N U T, 0, 0, 0',
	X =  119.242  mm,	Y =   -658.431  mm,	Z =   -267.000  mm,
	W =  90.000 deg,	P =   0.000 deg,	R =   90.000 deg
};
P[415]{
   GP1:
	UF : 0, UT : 6,		CONFIG : 'N U T, 0, 0, 0',
	X =  105.283  mm,	Y =   -666.502  mm,	Z =   -261.779  mm,
	W =  90.000 deg,	P =   0.000 deg,	R =   90.000 deg
};
P[416]{
   GP1:
	UF : 0, UT : 6,		CONFIG : 'N U T, 0, 0, 0',
	X =  100.725  mm,	Y =   -669.113  mm,	Z =   -247.571  mm,
	W =  90.000 deg,	P =   0.000 deg,	R =   90.000 deg
};
P[417]{
   GP1:
	UF : 0, UT : 6,		CONFIG : 'N U T, 0, 0, 0',
	X =  181.626  mm,	Y =   -622.663  mm,	Z =   -267.000  mm,
	W =  90.000 deg,	P =   0.000 deg,	R =   90.000 deg
};
P[418]{
   GP1:
	UF : 0, UT : 6,		CONFIG : 'N U T, 0, 0, 0',
	X =  202.296  mm,	Y =   -610.639  mm,	Z =   -267.000  mm,
	W =  90.000 deg,	P =   0.000 deg,	R =   90.000 deg
};
P[419]{
   GP1:
	UF : 0, UT : 6,		CONFIG : 'N U T, 0, 0, 0',
	X =  285.424  mm,	Y =   -562.629  mm,	Z =   -267.000  mm,
	W =  90.000 deg,	P =   0.000 deg,	R =   90.000 deg
};
P[420]{
   GP1:
	UF : 0, UT : 6,		CONFIG : 'N U T, 0, 0, 0',
	X =  327.144  mm,	Y =   -538.570  mm,	Z =   -267.000  mm,
	W =  90.000 deg,	P =   0.000 deg,	R =   90.000 deg
};
P[421]{
   GP1:
	UF : 0, UT : 6,		CONFIG : 'N U T, 0, 0, 0',
	X =  348.067  mm,	Y =   -526.432  mm,	Z =   -267.000  mm,
	W =  90.000 deg,	P =   0.000 deg,	R =   90.000 deg
};
P[422]{
   GP1:
	UF : 0, UT : 6,		CONFIG : 'N U T, 0, 0, 0',
	X =  368.908  mm,	Y =   -514.472  mm,	Z =   -267.000  mm,
	W =  90.000 deg,	P =   0.000 deg,	R =   90.000 deg
};
P[423]{
   GP1:
	UF : 0, UT : 6,		CONFIG : 'N U T, 0, 0, 0',
	X =  431.180  mm,	Y =   -478.495  mm,	Z =   -267.000  mm,
	W =  90.000 deg,	P =   0.000 deg,	R =   90.000 deg
};
P[424]{
   GP1:
	UF : 0, UT : 6,		CONFIG : 'N U T, 0, 0, 0',
	X =  452.044  mm,	Y =   -466.496  mm,	Z =   -267.000  mm,
	W =  90.000 deg,	P =   0.000 deg,	R =   90.000 deg
};
P[425]{
   GP1:
	UF : 0, UT : 6,		CONFIG : 'N U T, 0, 0, 0',
	X =  472.491  mm,	Y =   -454.921  mm,	Z =   -267.000  mm,
	W =  90.000 deg,	P =   0.000 deg,	R =   90.000 deg
};
P[426]{
   GP1:
	UF : 0, UT : 6,		CONFIG : 'N U T, 0, 0, 0',
	X =  514.312  mm,	Y =   -430.494  mm,	Z =   -267.000  mm,
	W =  90.000 deg,	P =   0.000 deg,	R =   90.000 deg
};
P[427]{
   GP1:
	UF : 0, UT : 6,		CONFIG : 'N U T, 0, 0, 0',
	X =  595.347  mm,	Y =   -383.642  mm,	Z =   -263.820  mm,
	W =  90.000 deg,	P =   0.000 deg,	R =   90.000 deg
};
P[428]{
   GP1:
	UF : 0, UT : 6,		CONFIG : 'N U T, 0, 0, 0',
	X =  602.785  mm,	Y =   -379.410  mm,	Z =   -247.535  mm,
	W =  90.000 deg,	P =   0.000 deg,	R =   90.000 deg
};
P[429]{
   GP1:
	UF : 0, UT : 6,		CONFIG : 'N U T, 0, 0, 0',
	X =  588.417  mm,	Y =   -415.081  mm,	Z =   -267.000  mm,
	W =  90.000 deg,	P =   0.000 deg,	R =   90.000 deg
};
P[430]{
   GP1:
	UF : 0, UT : 6,		CONFIG : 'N U T, 0, 0, 0',
	X =  546.794  mm,	Y =   -439.123  mm,	Z =   -267.000  mm,
	W =  90.000 deg,	P =   0.000 deg,	R =   90.000 deg
};
P[431]{
   GP1:
	UF : 0, UT : 6,		CONFIG : 'N U T, 0, 0, 0',
	X =  526.084  mm,	Y =   -451.298  mm,	Z =   -267.000  mm,
	W =  90.000 deg,	P =   0.000 deg,	R =   90.000 deg
};
P[432]{
   GP1:
	UF : 0, UT : 6,		CONFIG : 'N U T, 0, 0, 0',
	X =  505.440  mm,	Y =   -463.154  mm,	Z =   -267.000  mm,
	W =  90.000 deg,	P =   0.000 deg,	R =   90.000 deg
};
P[433]{
   GP1:
	UF : 0, UT : 6,		CONFIG : 'N U T, 0, 0, 0',
	X =  484.469  mm,	Y =   -475.263  mm,	Z =   -267.000  mm,
	W =  90.000 deg,	P =   0.000 deg,	R =   90.000 deg
};
P[434]{
   GP1:
	UF : 0, UT : 6,		CONFIG : 'N U T, 0, 0, 0',
	X =  463.919  mm,	Y =   -487.210  mm,	Z =   -267.000  mm,
	W =  90.000 deg,	P =   0.000 deg,	R =   90.000 deg
};
P[435]{
   GP1:
	UF : 0, UT : 6,		CONFIG : 'N U T, 0, 0, 0',
	X =  422.036  mm,	Y =   -511.261  mm,	Z =   -267.000  mm,
	W =  90.000 deg,	P =   0.000 deg,	R =   90.000 deg
};
P[436]{
   GP1:
	UF : 0, UT : 6,		CONFIG : 'N U T, 0, 0, 0',
	X =  339.103  mm,	Y =   -559.192  mm,	Z =   -267.000  mm,
	W =  90.000 deg,	P =   0.000 deg,	R =   90.000 deg
};
P[437]{
   GP1:
	UF : 0, UT : 6,		CONFIG : 'N U T, 0, 0, 0',
	X =  297.242  mm,	Y =   -583.446  mm,	Z =   -267.000  mm,
	W =  90.000 deg,	P =   0.000 deg,	R =   90.000 deg
};
P[438]{
   GP1:
	UF : 0, UT : 6,		CONFIG : 'N U T, 0, 0, 0',
	X =  276.720  mm,	Y =   -595.296  mm,	Z =   -267.000  mm,
	W =  90.000 deg,	P =   0.000 deg,	R =   90.000 deg
};
P[439]{
   GP1:
	UF : 0, UT : 6,		CONFIG : 'N U T, 0, 0, 0',
	X =  172.655  mm,	Y =   -655.063  mm,	Z =   -267.000  mm,
	W =  90.000 deg,	P =   0.000 deg,	R =   90.000 deg
};
P[440]{
   GP1:
	UF : 0, UT : 6,		CONFIG : 'N U T, 0, 0, 0',
	X =  117.400  mm,	Y =   -687.095  mm,	Z =   -261.540  mm,
	W =  90.000 deg,	P =   0.000 deg,	R =   90.000 deg
};
P[441]{
   GP1:
	UF : 0, UT : 6,		CONFIG : 'N U T, 0, 0, 0',
	X =  112.757  mm,	Y =   -690.007  mm,	Z =   -247.361  mm,
	W =  90.000 deg,	P =   0.000 deg,	R =   90.000 deg
};
P[442]{
   GP1:
	UF : 0, UT : 6,		CONFIG : 'N U T, 0, 0, 0',
	X =  131.322  mm,	Y =   -679.608  mm,	Z =   -266.984  mm,
	W =  90.000 deg,	P =   0.000 deg,	R =   90.000 deg
};
P[443]{
   GP1:
	UF : 0, UT : 6,		CONFIG : 'N U T, 0, 0, 0',
	X =  152.053  mm,	Y =   -667.547  mm,	Z =   -267.000  mm,
	W =  90.000 deg,	P =   0.000 deg,	R =   90.000 deg
};
P[444]{
   GP1:
	UF : 0, UT : 6,		CONFIG : 'N U T, 0, 0, 0',
	X =  193.668  mm,	Y =   -643.265  mm,	Z =   -267.000  mm,
	W =  90.000 deg,	P =   0.000 deg,	R =   90.000 deg
};
P[445]{
   GP1:
	UF : 0, UT : 6,		CONFIG : 'N U T, 0, 0, 0',
	X =  214.514  mm,	Y =   -631.245  mm,	Z =   -267.000  mm,
	W =  90.000 deg,	P =   0.000 deg,	R =   90.000 deg
};
P[446]{
   GP1:
	UF : 0, UT : 6,		CONFIG : 'N U T, 0, 0, 0',
	X =  235.389  mm,	Y =   -619.350  mm,	Z =   -267.000  mm,
	W =  90.000 deg,	P =   0.000 deg,	R =   90.000 deg
};
P[447]{
   GP1:
	UF : 0, UT : 6,		CONFIG : 'N U T, 0, 0, 0',
	X =  255.994  mm,	Y =   -607.455  mm,	Z =   -267.000  mm,
	W =  90.000 deg,	P =   0.000 deg,	R =   90.000 deg
};
P[448]{
   GP1:
	UF : 0, UT : 6,		CONFIG : 'N U T, 0, 0, 0',
	X =  318.478  mm,	Y =   -571.205  mm,	Z =   -267.000  mm,
	W =  90.000 deg,	P =   0.000 deg,	R =   90.000 deg
};
P[449]{
   GP1:
	UF : 0, UT : 6,		CONFIG : 'N U T, 0, 0, 0',
	X =  359.874  mm,	Y =   -547.412  mm,	Z =   -267.000  mm,
	W =  90.000 deg,	P =   0.000 deg,	R =   90.000 deg
};
P[450]{
   GP1:
	UF : 0, UT : 6,		CONFIG : 'N U T, 0, 0, 0',
	X =  380.714  mm,	Y =   -535.318  mm,	Z =   -267.000  mm,
	W =  90.000 deg,	P =   0.000 deg,	R =   90.000 deg
};
P[451]{
   GP1:
	UF : 0, UT : 6,		CONFIG : 'N U T, 0, 0, 0',
	X =  401.420  mm,	Y =   -523.311  mm,	Z =   -267.000  mm,
	W =  90.000 deg,	P =   0.000 deg,	R =   90.000 deg
};
P[452]{
   GP1:
	UF : 0, UT : 6,		CONFIG : 'N U T, 0, 0, 0',
	X =  442.842  mm,	Y =   -499.473  mm,	Z =   -267.000  mm,
	W =  90.000 deg,	P =   0.000 deg,	R =   90.000 deg
};
P[453]{
   GP1:
	UF : 0, UT : 6,		CONFIG : 'N U T, 0, 0, 0',
	X =  567.532  mm,	Y =   -427.491  mm,	Z =   -267.000  mm,
	W =  90.000 deg,	P =   0.000 deg,	R =   90.000 deg
};
P[454]{
   GP1:
	UF : 0, UT : 6,		CONFIG : 'N U T, 0, 0, 0',
	X =  607.299  mm,	Y =   -404.690  mm,	Z =   -263.704  mm,
	W =  90.000 deg,	P =   0.000 deg,	R =   90.000 deg
};
P[455]{
   GP1:
	UF : 0, UT : 6,		CONFIG : 'N U T, 0, 0, 0',
	X =  614.870  mm,	Y =   -400.316  mm,	Z =   -247.365  mm,
	W =  90.000 deg,	P =   0.000 deg,	R =   90.000 deg
};
P[456]{
   GP1:
	UF : 0, UT : 6,		CONFIG : 'N U T, 0, 0, 0',
	X =  126.228  mm,	Y =   -698.464  mm,	Z =   -257.879  mm,
	W =  90.000 deg,	P =   0.000 deg,	R =   90.000 deg
};
P[457]{
   GP1:
	UF : 0, UT : 6,		CONFIG : 'N U T, 0, 0, 0',
	X =  611.742  mm,	Y =   -420.008  mm,	Z =   -260.454  mm,
	W =  90.000 deg,	P =   0.000 deg,	R =   90.000 deg
};
P[458]{
   GP1:
	UF : 0, UT : 6,		CONFIG : 'N U T, 0, 0, 0',
	X =  596.961  mm,	Y =   -429.669  mm,	Z =   -262.179  mm,
	W =  90.000 deg,	P =   0.000 deg,	R =   90.000 deg
};
P[459]{
   GP1:
	UF : 0, UT : 6,		CONFIG : 'N U T, 0, 0, 0',
	X =  576.044  mm,	Y =   -441.874  mm,	Z =   -262.054  mm,
	W =  90.000 deg,	P =   0.000 deg,	R =   90.000 deg
};
P[460]{
   GP1:
	UF : 0, UT : 6,		CONFIG : 'N U T, 0, 0, 0',
	X =  555.108  mm,	Y =   -453.956  mm,	Z =   -261.994  mm,
	W =  90.000 deg,	P =   0.000 deg,	R =   90.000 deg
};
P[461]{
   GP1:
	UF : 0, UT : 6,		CONFIG : 'N U T, 0, 0, 0',
	X =  534.413  mm,	Y =   -465.820  mm,	Z =   -262.219  mm,
	W =  90.000 deg,	P =   0.000 deg,	R =   90.000 deg
};
P[462]{
   GP1:
	UF : 0, UT : 6,		CONFIG : 'N U T, 0, 0, 0',
	X =  513.842  mm,	Y =   -477.685  mm,	Z =   -262.204  mm,
	W =  90.000 deg,	P =   0.000 deg,	R =   90.000 deg
};
P[463]{
   GP1:
	UF : 0, UT : 6,		CONFIG : 'N U T, 0, 0, 0',
	X =  492.820  mm,	Y =   -489.868  mm,	Z =   -262.135  mm,
	W =  90.000 deg,	P =   0.000 deg,	R =   90.000 deg
};
P[464]{
   GP1:
	UF : 0, UT : 6,		CONFIG : 'N U T, 0, 0, 0',
	X =  472.126  mm,	Y =   -501.925  mm,	Z =   -261.931  mm,
	W =  90.000 deg,	P =   0.000 deg,	R =   90.000 deg
};
P[465]{
   GP1:
	UF : 0, UT : 6,		CONFIG : 'N U T, 0, 0, 0',
	X =  451.619  mm,	Y =   -513.617  mm,	Z =   -262.206  mm,
	W =  90.000 deg,	P =   0.000 deg,	R =   90.000 deg
};
P[466]{
   GP1:
	UF : 0, UT : 6,		CONFIG : 'N U T, 0, 0, 0',
	X =  430.546  mm,	Y =   -525.817  mm,	Z =   -262.113  mm,
